(* CODESYS project METIS_CRYO.library
   Version: 0.1.1
   Title: METIS Cryo PLC
   Author: Muhammad Salman
   Placeholder: METIS Cryo PLC
   Company: KU Leuven

Project tree, tasks and I/O mapping:
  libraries: CmpBitmapPool, * (System); ESO Cryo HMI Library, * (ESO); ESO LDC Comm Common Library, * (ESO); ESO LDC Comm Tcp Library, * (ESO); ESO LDC Control Library, * (ESO); ESO LDC Cryo Library, * (ESO); ESO LDC Timer Library, * (ESO); FloatingPointUtils, * (System); METIS CCU, * (KU Leuven); METIS Fuse Library, * (KU Leuven); Recipe Management, * (System); Tc2_ControllerToolbox, * (Beckhoff Automation GmbH); Tc2_Standard, * (Beckhoff Automation GmbH); Tc2_System, * (Beckhoff Automation GmbH); Tc2_Utilities, * (Beckhoff Automation GmbH); Tc2_XmlDataSrv, * (Beckhoff Automation GmbH); Tc3_Module, * (Beckhoff Automation GmbH); VisuDialogs, * (System); VisuSymbols, * (System)
  DUTs/
    Enumerators/
      Actuators/
      Ctrl_Valves/
        data type E_METIS_CRYO_CTRL_VALVE_STATE
        data type E_METIS_CRYO_CTRL_VALVE_TYPE
      Heaters/
        data type E_METIS_CRYO_HEATER_STATE
        data type E_METIS_CRYO_HEATER_TYPE
        data type E_METIS_PWM_HEATER_CTRL
      LN2_Level/
        data type E_LN2_LEVEL_CTRL_STATE
      Routines/
        Anti_Fogging/
          data type E_ANTI_FOGGING_MODE
          data type E_MET_CRYO_ANTI_FOGGING_STATE
        Cool_Down/
          data type E_MET_CRYO_COOLDOWN_PRESSURES
          data type E_MET_CRYO_COOLDOWN_STATE
          data type E_MET_CRYO_COOLDOWN_SYS_STATE
          data type E_MET_CRYO_COOLDOWN_VALVES
          data type E_MET_CRYO_LN2_FILLING_STATE
        Re_Generation/
          data type E_MET_CRYO_RE_GENERATION_STATE
        Venting/
          data type E_MET_CRYO_VENTING_PRESSURES
          data type E_MET_CRYO_VENTING_STATE
          data type E_MET_CRYO_VENTING_SYS_STATE
          data type E_MET_CRYO_VENTING_VALVES
        WarmUp/
          data type E_MET_CRYO_WARMUP_STATE
      Sensors/
        Base_Sensor/
          data type E_METIS_SENSOR_SOURCE
          data type E_METIS_SENSOR_TYPE
        LN2_Level_Sensor/
          data type E_METIS_CRYO_LN2_SENSOR_LEVELS
        Temperature Sensor/
          data type E_METIS_LAKE_SHORE_TYPE
          data type E_METIS_TEMP_VOTE_METHOD
      System/
        data type E_METIS_CRYO_CTRL_CMD
        data type E_METIS_CRYO_CTRL_STATE
    Structures/
      Actuators/
      Base_Sensor/
        data type T_METIS_SENSOR_BASE_STATUS
      Ctrl_Valves/
        data type T_METIS_CTRL_VALVE_CFG
        data type T_METIS_CTRL_VALVE_CTRL
        data type T_METIS_CTRL_VALVE_IO_ANTI_FOG_BLOWER
        data type T_METIS_CTRL_VALVE_IO_IMG_CFO_PRECOOLING
        data type T_METIS_CTRL_VALVE_STAT
      Error_Handeling/
        data type T_METIS_CRYO_ERROR_STATUS
      Heaters/
        METIS_HEATER/
          data type T_METIS_HEATER_CFG
          data type T_METIS_HEATER_CTRL
          data type T_METIS_HEATER_IO_CPAU60
          data type T_METIS_HEATER_IO_CXWUI60
          data type T_METIS_HEATER_IO_EL95X1
          data type T_METIS_HEATER_IO_PWM
          data type T_METIS_HEATER_STAT
        data type T_METIS_CRYO_HEATER_CTRL
        data type T_METIS_CRYO_HEATER_STATUS
      LN2_Level_Ctrl/
        data type T_LN2_LEVEL_CTRL_CFG
        data type T_LN2_LEVEL_CTRL_CTRL
      PID_Control/
        Generic/
          data type E_METIS_CTRL_MODE
          data type E_METIS_CTRL_SETPOINT_SWITCH
          data type T_METIS_CTRL_LOOP_CFG
          data type T_METIS_CTRL_LOOP_CTRL
          data type T_METIS_CTRL_LOOP_STAT
          text list TEXTLIST_METIS_CTRL_MODE
        data type T_METIS_CTRL_BASE_CFG
        data type T_METIS_CTRL_BASE_CTRL
        data type T_METIS_CTRL_BASE_STAT
      RAMP/
        data type T_METIS_CTRL_RAMP_CTRL
        data type T_METIS_CTRL_RAMP_STAT
      Routines/
        Anti_Fogging/
          data type T_MET_CRYO_ANTI_FOGGING_CTRL
          data type T_MET_CRYO_ANTI_FOGGING_STAT
        Cool_Down/
          data type T_MET_CRYO_COOLDOWN_CFG
          data type T_MET_CRYO_COOLDOWN_CTRL
          data type T_MET_CRYO_COOLDOWN_STAT
          data type T_MET_CRYO_COOLDOWN_SYS_INPUT
          data type T_MET_CRYO_COOLDOWN_SYSTEM_STATUS
        Evacuation/
          data type T_MET_CRYO_EVACUATION_CTRL
          data type T_MET_CRYO_EVACUATION_STAT
        Re_Generation/
          data type T_MET_CRYO_RE_GENERATION_CTRL
          data type T_MET_CRYO_RE_GENERATION_STAT
        Venting/
          data type T_MET_CRYO_VENTING_CFG
          data type T_MET_CRYO_VENTING_CTRL
          data type T_MET_CRYO_VENTING_STAT
          data type T_MET_CRYO_VENTING_SYS_INPUT
          data type T_MET_CRYO_VENTING_SYSTEM_STATUS
        WarmUp/
          data type T_MET_CRYO_WARMUP_CTRL
          data type T_MET_CRYO_WARMUP_STAT
      Sensors/
        LN2_Level_Sensor/
          data type T_METIS_CRYO_LN2_LEVEL_CFG
          data type T_METIS_CRYO_LN2_LEVEL_STATUS
      System/
        data type T_METIS_CRYO_CFG
        data type T_METIS_CRYO_CTRL
        data type T_METIS_CRYO_DEBUG
        data type T_METIS_CRYO_EVENTS
        data type T_METIS_CRYO_INTERLOCKS
        data type T_METIS_CRYO_STAT
        data type T_METIS_CRYO_TRIGGERS
      Temp_Sensor/
        data type T_METIS_DT670_TEMP_SENSOR_STATUS
      Temp_Voter/
        data type T_HMI_METIS_TEMP_VOTER_CTRL
        data type T_HMI_METIS_TEMP_VOTER_STAT
        data type T_METIS_CRYO_TEMP_VOTE_STATUS
        data type T_METIS_TEMP_VOTE_CFG
        data type T_METIS_TEMP_VOTERS_CTRL
      Temperature/
        data type E_ALL_METIS_TEMPERATURES
        data type T_METIS_TEMPERATURE_STATUS
  GVLs/
  HMI/
    DUTs/
      Cryo_Devices/
        Temperatures/
          data type E_HMI_TEMP_TABS
        data type E_HMI_PUMPS_TABS
      Subsystems/
        CFO/
          data type E_HMI_CFO_TABS
        CRY/
          Components/
            data type E_HMI_CRY_HEATER_TABS
            data type E_HMI_CRY_TC_TABS
          data type E_HMI_CRY_TABS
        ICS/
          data type E_HMI_ICS_TABS
        IMG/
          Components/
            data type E_HMI_IMG_HEATER_TABS
            data type E_HMI_IMG_TC_TABS
          data type E_HMI_IMG_TABS
        LMS/
          data type E_HMI_LMS_TABS
        SCA/
          Components/
            data type E_HMI_SCA_HEATER_TABS
            data type E_HMI_SCA_TC_TABS
          data type E_HMI_SCA_TABS
      System/
        data type E_HMI_TABS
      Util/
        data type E_HMI_COLORS
        data type E_HMI_VOTER_TABS
        data type T_ECAT_MODULE
        data type T_HMI_COLORS
    POUs/
      Cryo-Routines/
        Anti-Fogging/
          function block FB_HMI_ANTI_FOGGING [ST]
        Cool-Down/
          function block FB_HMI_COOL_DOWN [ST]
        Evacuation/
          function block FB_HMI_EVACUATION [ST]
        Power-Outage/
          function block FB_HMI_POWER_OUTAGE [ST]
        Regeneration/
          function block FB_HMI_REGENERATION [ST]
        Venting/
          function block FB_HMI_VENTING [ST]
        Warm-Up/
          function block FB_HMI_WARM_UP [ST]
      Devices/
        Cabinets/
          function block FB_HMI_CABINETS [ST]
          function block FB_HMI_CCU [ST]
        Control_Loops/
          function block FB_HMI_CONTROL_LOOPS [ST]
          function block FB_HMI_METIS_CTRL_TEMPERATURE [ST]
        Control_Units/
          function block FB_HMI_CONTROL_UNITS [ST]
        Coolers/
          function block FB_HMI_COOLERS [ST]
        Detectors/
          function block FB_HMI_DETECTORS [ST]
        Heaters/
          function block FB_HMI_HEATERS [ST]
          function block FB_HMI_METIS_HEATER [ST]
        Lakeshores/
          function block FB_HMI_LAKESHORE [ST]
        Pressures/
          function block FB_HMI_PRESSURES [ST]
        Pumps/
          function block FB_HMI_PUMPS [ST]
          function block FB_HMI_RP_BRANCH_A [ST]
          function block FB_HMI_RP_BRANCH_B [ST]
          function block FB_HMI_TP_BRANCH_A [ST]
          function block FB_HMI_TP_BRANCH_B [ST]
        RH/
          function block FB_HMI_METIS_RH_SENSOR [ST]
        Temperatures/
          Components/
            function block FB_HMI_TEMP_VOTERS [ST]
          function block FB_HMI_TEMPERATURES [ST]
        Valves/
          function block FB_HMI_VALVES [ST]
        Voters/
          function block FB_HMI_VOTER [ST]
        function block FB_HMI_DEVICES [ST]
      Events/
        function block FB_HMI_EVENTS [ST]
      ICS_Interlocks/
        function block FB_HMI_ICS_INTERLOCKS [ST]
      Services/
        Status/
          function F_HMI_BUSY_TO_COLOR [ST]
          function F_HMI_HEALTH_BUSY_TO_COLOR [ST]
          function F_HMI_HEALTH_TO_COLOR [ST]
          function block FB_HMI_BUSY_STATUS [ST]
          function block FB_HMI_HEALTH_STATUS [ST]
          function block FB_HMI_STATUS [ST]
        function block FB_HMI_SERVICES [ST]
        function block FB_HMI_SERVICES_TIME [ST]
      Subsystems/
        CFO/
          Components/
            function block FB_HMI_CFO_HEATERS [ST]
            function block FB_HMI_CFO_TCTRL [ST]
            function block FB_HMI_CFO_TEMPERATURES [ST]
            function block FB_HMI_CFO_VOTERS [ST]
          function block FB_HMI_CFO [ST]
        CRY/
          Components/
            function block FB_HMI_CRY_HEATERS [ST]
            function block FB_HMI_CRY_LN2CTRL [ST]
            function block FB_HMI_CRY_RH [ST]
            function block FB_HMI_CRY_TCTRL [ST]
            function block FB_HMI_CRY_TEMPERATURES [ST]
            function block FB_HMI_CRY_VOTERS [ST]
          function block FB_HMI_CRY [ST]
        ICS/
          function block FB_HMI_ICS [ST]: M_UpdateConfigsColor
        IMG/
          Components/
            function block FB_HMI_IMG_HEATERS [ST]
            function block FB_HMI_IMG_TCTRL [ST]
            function block FB_HMI_IMG_TEMPERATURES [ST]
            function block FB_HMI_IMG_VOTERS [ST]
          function block FB_HMI_IMG [ST]
        LMS/
          Components/
            function block FB_HMI_LMS_HEATERS [ST]
            function block FB_HMI_LMS_TCTRL [ST]
            function block FB_HMI_LMS_TEMPERATURES [ST]
            function block FB_HMI_LMS_VOTERS [ST]
          function block FB_HMI_LMS [ST]
        SCA/
          Components/
            function block FB_HMI_SCA_HEATERS [ST]
            function block FB_HMI_SCA_TCTRL [ST]
            function block FB_HMI_SCA_TEMPERATURES [ST]
            function block FB_HMI_SCA_VOTERS [ST]
          function block FB_HMI_SCA [ST]
      Util/
        Button/
          function block FB_HMI_BUTTON [ST]: FB_init, M_SetIconName
        Component/
          function block FB_HMI_COMPONENT [ST]: M_UpdateStatusColor
        Functions/
          function F_GetConnectionColor [ST]
          function F_GetConnectionString [ST]
        function block FB_HMI_BACK [ST]
        function block FB_HMI_CRYO_SIM [ST]
    VISUs/
      Cryo_Devices/
        Cabinets/
          visualisation VISU_HMI_CABINETS
        Control_Loops/
          visualisation VISU_HMI_CONTROL_LOOPS
        Control_Units/
          visualisation VISU_HMI_CONTROL_UNITS
        Coolers/
          visualisation VISU_HMI_COOLERS
        Detectors/
          visualisation VISU_HMI_DETECTORS
        Heaters/
          visualisation VISU_HMI_HEATERS
        Pressures/
          visualisation VISU_HMI_PRESSURES
        Pumps/
          visualisation VISU_HMI_PUMPS
          visualisation VISU_HMI_RP_BRANCH_A
          visualisation VISU_HMI_RP_BRANCH_B
          visualisation VISU_HMI_TP_BRANCH_A
          visualisation VISU_HMI_TP_BRANCH_B
        Temperatures/
          Components/
            visualisation VISU_HMI_SYSTEM_VOTERS
          visualisation VISU_HMI_TEMPERATURES
        Valves/
          visualisation VISU_HMI_VALVES
        visualisation VISU_HMI_DEVICES_DIALOG
      Cryo-Routines/
        Anti-Fogging/
          visualisation VISU_HMI_ANTI_FOGGING
        Cool-Down/
          visualisation VISU_HMI_COOL_DOWN
        Evacuation/
          visualisation VISU_HMI_EVACUATION
        Power-Outage/
          visualisation VISU_HMI_POWER_OUTAGE
        Regeneration/
          visualisation VISU_HMI_REGENERATION
          visualisation VISU_REGENERATION_CTRL
          visualisation VISU_SORPTION_HEATER
          visualisation VISU_SORPTION_TEMP_VOTE
        Venting/
          visualisation VISU_HMI_VENTING
        Warm-Up/
          visualisation VISU_HMI_WARM_UP
      Events/
        visualisation VISU_HMI_EVENTS
      GUIs/
        visualisation GUI_LN2_LEVEL_CTRL
        visualisation GUI_MANUAL_CONTROL
        visualisation GUI_METIS_EVACUATION
        visualisation VISU_HMI_FUSE_HMI
      Home/
        visualisation VISU_HMI_HOME
      ICS_Interlocks/
        visualisation VISU_HMI_ICS_INTERLOCKS
      Services/
        visualisation VISU_HMI_SERVICES
      SIM_GUIs/
        visualisation GUI_Pressures_1
        visualisation GUI_SIM_PRESSURES
        visualisation GUI_SIM_SYSTEM_STATE
        visualisation GUI_SIM_TEMPERATURES
        visualisation VISU_SIM_PRESS_AND_TEMPS
      Subsystems/
        CFO/
          Components/
          visualisation VISU_HMI_CFO
        CRY/
          Components/
            visualisation VISU_HMI_CRY_HEATERS
            visualisation VISU_HMI_CRY_LN2_LEVEL_CONTROL
            visualisation VISU_HMI_CRY_RH
            visualisation VISU_HMI_CRY_TCTRL
            visualisation VISU_HMI_CRY_TEMPERATURES
            visualisation VISU_HMI_CRY_VOTERS
          visualisation VISU_HMI_CRY
        ICS/
          Components/
            visualisation VISU_HMI_ICS_CCU_CONFIGS
            visualisation VISU_HMI_ICS_CCUS_CONFIGS
          visualisation VISU_HMI_ICS
        IMG/
          Components/
            visualisation VISU_HMI_IMG_HEATERS
            visualisation VISU_HMI_IMG_TC
            visualisation VISU_HMI_IMG_TEMPERATURES
            visualisation VISU_HMI_IMG_VOTERS
          visualisation VISU_HMI_IMG
        LMS/
          visualisation VISU_HMI_LMS
        SCA/
          Components/
            visualisation VISU_HMI_SCA_HEATERS
            visualisation VISU_HMI_SCA_TC
            visualisation VISU_HMI_SCA_TEMPERATURES
            visualisation VISU_HMI_SCA_VOTERS
          visualisation VISU_HMI_SCA
      Templates/
        visualisation ARCHIVED_TEMPLATE_MAIN_FSM_1
        visualisation GUI_EVAC_BRANCH_A_1
        visualisation GUI_Events
        visualisation GUI_RP_PUMPS
        visualisation GUI_TEMPLATE_LAKESHORE_336_TCP
        visualisation GUI_TP_PUMPS
        image pool ImagePool_1
        visualisation Sim_LN2_Ctrl_inputs
        visualisation TEMPLATE_AMBIENT_PRESSURE_READING
        visualisation TEMPLATE_BACKGROUND_LEVEL_2
        visualisation TEMPLATE_BACKGROUND_LEVEL_3
        visualisation TEMPLATE_BINARY_VALVES
        visualisation TEMPLATE_CRYO_SENSOR_TEMPERATURE
        visualisation TEMPLATE_EVACUATION
        visualisation TEMPLATE_HEATER_CPAU60
        visualisation TEMPLATE_HEATER_CXWUI60
        visualisation TEMPLATE_HEATER_PWM_CTRL
        visualisation TEMPLATE_LN2_LEVEL_SENSOR_AND_CTRL
        visualisation TEMPLATE_MAIN_FSM
        visualisation TEMPLATE_METIS_CMD_OVERRIDE
        visualisation TEMPLATE_METIS_CONTROL_VALVE
        visualisation TEMPLATE_METIS_CRYO_CPA
        visualisation TEMPLATE_METIS_CRYO_CPAU60_PID_CTRL
        visualisation TEMPLATE_METIS_CRYO_PWM_PID_CTRL
        visualisation TEMPLATE_METIS_CTRL_TEMPERATURE
        visualisation TEMPLATE_METIS_CTRL_TEMPERATURE_MPIA
        visualisation TEMPLATE_METIS_CTRL_TEMPERATURE_SIMPLIFIED
        visualisation TEMPLATE_METIS_HEATER
        visualisation TEMPLATE_METIS_HEATER_SIMPLIFIED
        visualisation TEMPLATE_PRESSURE_READING
        visualisation TEMPLATE_RESET_VALVES
        visualisation TEMPLATE_TEMP_SENSOR_VALUE_ONLY
        visualisation TEMPLATE_TEMPERATURE_VOTE
      Util/
        Button/
          image pool VISU_HMI_BUTTON_IMAGES
          visualisation VISU_HMI_ROUTINES_BUTTON
          visualisation VISU_HMI_SUBSUBSYSTEM_BUTTON
          visualisation VISU_HMI_SUBSYSTEM_BUTTON
          visualisation VISU_HMI_SYSTEM_BUTTON
        image pool ICONS_IMAGE_POOL
    program PRG_HMI [ST]: M_TrackPreviousTab, M_UpdateStatus
    visualisation VISU_HMI
  00000000-0000-0000-0000-000000000000|IMAGES\Evacuation_schematics.png
  00000000-0000-0000-0000-000000000000|IMAGES\METIS_Cryo_FSM.png
  00000000-0000-0000-0000-000000000000|HMI\Images\Button\home.png
  00000000-0000-0000-0000-000000000000|HMI\Images\Button\cover.png
  00000000-0000-0000-0000-000000000000|HMI\Images\Button\m1.png
  00000000-0000-0000-0000-000000000000|HMI\Images\Button\m3.png
  00000000-0000-0000-0000-000000000000|HMI\Images\Button\services.png
  00000000-0000-0000-0000-000000000000|HMI\Images\Button\telemetry.png
  00000000-0000-0000-0000-000000000000|HMI\Images\Button\m2.png
  00000000-0000-0000-0000-000000000000|HMI\Images\Button\hydraulics.png
  00000000-0000-0000-0000-000000000000|HMI\Images\Button\safety.png
  00000000-0000-0000-0000-000000000000|HMI\Images\Button\axes.png
  00000000-0000-0000-0000-000000000000|HMI\Images\Button\dome.png
  00000000-0000-0000-0000-000000000000|HMI\Images\Button\Events.png
  00000000-0000-0000-0000-000000000000|HMI\Images\Button\subsystems.png
  00000000-0000-0000-0000-000000000000|HMI\Images\Button\interlock.png
  00000000-0000-0000-0000-000000000000|Images\metis_logo_white.png
  00000000-0000-0000-0000-000000000000|Images\metis_logo_color.png
  HMIWrapperFBs/
    function block FB_METIS_HMI_CRYO_TEMPERATURE_VOTE [ST]: M_ProcessInput, M_UpdateStatus
  IMAGES/
    Evacuation_schematics.png
  POUs/
    Control/
      Control/
        function block FB_METIS_CTRL_BASE [ST]: M_CheckErrors, M_Configure, M_ExecuteController, M_Read_Write_Config, M_Set_PID_Parameters, M_SetAutoMode, M_SetEngMode, M_SetManualMode, M_SetPermissionMode, M_SetRamp
        function block FB_METIS_CTRL_RAMP_GENERATOR [ST]: M_Configure, M_ExecuteController
        function block FB_METIS_CTRL_TEMPERATURE [ST]: M_ConfigReadingFinished, M_Configure, M_ExecuteController, M_ExecuteModes, M_Read_Write_Config, M_Set_SetPoint, M_SetDisable, M_SetEnable, M_Startup, M_UpdateAlarms, M_UpdateStatus, M_UpdateTempPointers
        function block FB_PWM_PID_CTRL [ST]
      Process/
        function block FB_FT1_SIM_PROCESS [ST]
      TCtrl/
        function block FB_METIS_TCTRL [ST]
    Devices/
      AmbientPressure/
        function block FB_METIS_AMBIENT_PRESSURE_SENSOR [ST]: M_SetStatus, M_SetStatus_CMR_361, M_SetStatus_MIPA_015A, M_SetStatus_PKR_250, M_SetStatus_PKR_360, M_SetStatus_WRG_D_NW25
      Base_Sensor/
        function block FB_METIS_SENSOR_BASE [ST]: M_GetRamp, M_ReadSensor, M_SetStatus, M_SetStatus_LS240
      CCU/
        function block FB_METIS_CCUS [ST]: M_Configure
      Control_Valves_Ctrl/
        function block FB_METIS_CONTROL_VALVE [ST]: M_Activity_Valve_Alarm, M_Activity_Valve_None, M_Activity_Valve_Normal, M_Configure, M_GetError, M_IsValveInError, M_Read_Write_Config, M_ReadInputs, M_ScaleInput, M_ScaleOutput, M_SetCtrlOutput, M_SetDisable, M_SetEnable, M_SetManualDisable, M_SetManualEnable, M_SetMode, M_SetStatus, M_UpdateActive, M_UpdateAlarms
      DigitalOutput/
        function block FB_METIS_DO [ST]: M_Configure, M_UpdateStatus
        data type T_METIS_DO_CTRL
        data type T_METIS_DO_STAT
      Heaters/
        Heater_Ctrl/
          function block FB_HEATER_CPAU60 [ST]: bIsActive, bIsInError, bIsNotActive, lrHeaterPower, M_Activate, M_Configure, M_DeActivate, M_GetHeaterPower, M_ReadInputs, M_ScaleInput, M_ScaleOutput, M_SetCtrlOutput, M_SetHeaterPower, M_SetManualInputFlag, M_SetStatus
          function block FB_HEATER_CXWUI60 [ST]: bIsActive, bIsInError, bIsNotActive, lrHeaterPower, M_Activate, M_Configure, M_DeActivate, M_GetHeaterPower, M_ReadInputs, M_ScaleInput, M_ScaleOutput, M_SetCtrlOutput, M_SetHeaterPower, M_SetManualInputFlag, M_SetStatus
          function block FB_HEATER_PWM [ST]: bIsActive, bIsInError, bIsNotActive, lrHeaterPower, M_Activate, M_DeActivate, M_GetHeaterPower, M_ReadInputs, M_ScaleInput, M_ScaleOutput, M_SetCtrlOutput, M_SetHeaterPower, M_SetManualInputFlag, M_SetStatus
          function block FB_METIS_HEATER [ST]: M_Configure, M_isHeaterInError, M_Read_Write_Config, M_ReadInputs, M_ScaleInput, M_ScaleOutput, M_SetCtrlOutput, M_SetDisable, M_SetEnable, M_SetMode, M_SetStatus, M_UpdateAlarms
          interface I_Heater: bIsActive, bIsInError, bIsNotActive, lrHeaterPower, M_Activate, M_DeActivate
        function block FB_METIS_HEATERS [ST]: M_ExecuteControllers
      LakeShore_336/
        function block FB_METIS_LAKESHORE_336_TCP [ST]: M_Configure, M_GetCommInitialised, M_GetCommStatus, M_SetTemperatureOutputs, M_UpdateStatus
        function block FB_METIS_LAKESHORES [ST]
      LN2_Level_Ctrl/
        function block FB_METIS_CRYO_LN2_LEVEL_CTRL [ST]: M_Activity_CheckPreConditions, M_Activity_EarlyRefilling, M_Activity_ErrorHandeling, M_Activity_Level_Monitoring, M_Check_LN2_Level, M_Configure, M_ExecuteControllers, M_FillingControl, M_HandleEvents, M_Read_Write_Config, M_ReadSensors, M_Reset, M_ResetValve, M_Set_LN2FillingFlag, M_StateMachine, M_UpdateAlarms, M_UpdateStatus
      LN2_Level_Sensor/
        function block FB_LN2_LEVEL_PT100_SENSOR [ST]
        function block FB_METIS_CRYO_LN2_SENSOR [ST]: M_ReadSensors, M_SetHeatersOutput, M_SetOutput, M_SetStatus
      PTC Cooler/
        function block FB_METIS_CRYO_CPA [ST]: M_CompressorRunning, M_HighPressureFlag, M_HighTemperatureFlag
      RH_Sensor/
        function block FB_METIS_RH [ST]
        function block FB_METIS_RH_DEWPOINT_CALC [ST]
        function block FB_METIS_RH_SENSOR [ST]: M_ReadSensor, M_SetStatus
        data type T_METIS_RH_SENSOR_STAT
      Temp_Sensor/
        function block FB_METIS_TEMP_SENSOR_DT670 [ST]: M_GetRamp, M_ReadSensor, M_SetSensorStatus_DT670_LS240, M_SetSensorStatus_DT670_LS336, M_SetSensorStatus_DT670_Ramp, M_SetSensorStatus_DT670_Voter, M_SetStatus, M_SetTemperature
        function block FB_SIM_TEMP_SENSOR_DT670 [ST]: M_Configure, M_ExecuteController
      Temp_Voter/
        function block FB_METIS_VOTER [ST]: bTempNotValid, bTempValid, lrRamp, lrTempK, M_ConfigReadingFinished, M_Configure, M_GetRamp, M_Read_Write_Config, M_SetPermissionMode, M_SetStatus, M_SetStatus_Average, M_SetStatus_FirstValid, M_SetStatus_Highest_Temperature, M_SetStatus_Lowest_Temperature, M_SetStatus_Median, M_SetStatus_XooY, M_UpdateAlarms, M_UpdateTempPointers
        function block FB_METIS_VOTER_COPY_for_new_HMI [ST]: bTempNotValid, bTempValid, lrRamp, lrTempK, M_ConfigReadingFinished, M_Configure, M_GetRamp, M_Read_Write_Config, M_SetPermissionMode, M_SetStatus, M_SetStatus_Average, M_SetStatus_FirstValid, M_SetStatus_Highest_Temperature, M_SetStatus_Lowest_Temperature, M_SetStatus_Median, M_SetStatus_XooY, M_UpdateTempPointers
        function block FB_METIS_VOTERS [ST]: M_ProcessHmi, M_ReadSensors
      Temperature/
        function block FB_METIS_TEMPERATURE [ST]
        function block FB_METIS_TEMPERATURES [ST]: M_ConfigSimTemperatures, M_Configure, M_GetTempSensorIndex, M_IsIgnoredTemperature, M_MaxMinAvrgTemperatures, M_ReadSensors, M_SetTemperatureSensor, M_UpdatePointer, M_UpdatePointers
    Functions/
      function F_TIME_HHMMSS [ST]
      function F_TON_TO_TIME_STRING [ST]
    Routines/
      AntiFogging/
        function block FB_METIS_CRYO_ANTI_FOGGING [ST]: M_Activity_AirBlowing, M_Activity_Alarm_Condition, M_Activity_Check_Preconditions, M_Activity_Error_Handling, M_Activity_Finished, M_Activity_Heating, M_Activity_None, M_Activity_Standard_Operation, M_Activity_Start_Anti_Fogging, M_Configure, M_Evaluate_DewPoint_State, M_ExecuteControllers, M_HandleEvents, M_SetError, M_Start_AntiFogging, M_StateMachine, M_Stop_AntiFogging, M_UpdateStatus
      CabinetControl/
        function block FB_METIS_CABINET_CTRL [ST]
      CoolDown/
        function block FB_METIS_CRYO_COOL_DOWN [ST]: M_Activity_Check_Preconditions, M_Activity_Cold_State, M_Activity_Cool_Down_Finished, M_Activity_Error_Handling, M_Activity_Finished, M_Activity_Keep_Cooling, M_Activity_None, M_Activity_Start_Cool_Down, M_Activity_Start_LN2_Filling, M_Activity_Start_PTCs, M_Activity_Start_Temp_Ctrl_PTC, M_Activity_Stop_LN2_Filling, M_Activity_Stop_PTCs, M_Activity_Stopping_Cool_Down, M_Check_Is_ReadyForOperation, M_Check_LN2_Filling_Status, M_Check_PTCs_Heater_Ctrl_Status, M_Check_PTCs_Status, M_Configure, M_ExecuteControllers, M_Get_ReadyForOperations, M_HandleEvents, M_HandleInterlocks, M_Manage_Early_Refilling, M_PermitEvacuationStop, M_ReadSensors, M_ResetValves, M_SetError, M_Simulated_Sens_Acts, M_Standalone_LN2_Filling, M_StateMachine, M_Stop_PTCs_During_WarmUP, M_UpdateStatus
      Evacuation/
        function block FB_CRYO_EVAC_BRANCH_A [ST]: M_Configure, M_ExecuteControllers, M_HandleInterlocks, M_ResetValves
        function block FB_CRYO_EVAC_BRANCH_B [ST]: M_Configure, M_ExecuteControllers, M_HandleInterlocks, M_ResetValves
        function block FB_METIS_CRYO_EVAC [ST]: M_AreAnyPumpsRunning, M_AreRoughingPumpRunning, M_AreTurboPumpsRunning, M_CheckBranchError, M_Configure, M_ExecuteControllers, M_HandleEvents, M_HandleInterlocks, M_ResetValves, M_SetAuto, M_SetError, M_Start_Evacuation, M_Stop_Evacuation, M_UpdateStatus
      PowerOutage/
        function block FB_METIS_CRYO_POWER_OUTAGE [ST]
      Regeneration/
        function block FB_METIS_CRYO_REGENERATION [ST]: M_Activity_Check_Preconditions, M_Activity_CoolDownSP, M_Activity_ErrorHandeling, M_Activity_Finished, M_Activity_KeepHeating, M_Activity_None, M_Activity_StartHeating, M_Configure, M_ExecuteControllers, M_HandleEvents, M_PermitEvacuationStop, M_SetError, M_StateMachine, M_UpdateStatus
      StopPowerOutage/
        function block FB_METIS_CRYO_STOP_POWER_OUTAGE [ST]
      Venting/
        function block FB_METIS_CRYO_VENTING [ST]: M_Activity_Check_Preconditions, M_Activity_ClosingValve, M_Activity_Error_Handling, M_Activity_None, M_Activity_OpeningValve, M_Activity_Prepare_For_Venting, M_Activity_Start_Venting, M_Activity_Stop_Venting, M_Activity_Venting_InProgress, M_AreVentingValvesClosed, M_Close_Venting_Valves, M_Configure, M_ExecuteControllers, M_HandleEvents, M_HandleInterlocks, M_IsVentingFinishedSuccessfully, M_Open_Venting_Valves, M_ReadSensors, M_ResetValves, M_SetError, M_StateMachine, M_UpdateStatus
      WarmUP/
        function block FB_METIS_CRYO_WARM_UP [ST]: M_Activity_Check_Preconditions, M_Activity_Error_Handling, M_Activity_Finished, M_Activity_Keep_Ramping_Up_Detectors, M_Activity_Keep_Warming_Up, M_Activity_None, M_Activity_Ramp_Up_Detectors_2, M_Activity_Start_Ramp_Up_CFO, M_Activity_Start_Ramp_Up_Detectors_1k, M_Activity_Start_Ramp_Up_IMG, M_Activity_Start_Ramp_Up_LMS, M_Activity_Start_Ramp_Up_Radiation_Shields, M_Activity_Start_Ramp_Up_SCAO, M_Activity_Start_Warm_Up, M_Activity_Stop_PTCs, M_Activity_Stopping_Warm_Up, M_AreWarmUpHeaterActive, M_CheckTCErrors, M_Configure, M_HandleEvents, M_HandleInterlocks, M_PermitEvacuationStop, M_PermitVenting, M_SetError, M_StateMachine, M_UpdateStatus
    Services/
      function block FB_SERVICES [ST]
    Simulation/
      function block FB_SIM_LN2_LEVEL_VALVES [ST]
      function block FB_SIM_LN2_SENSOR [ST]
      function block FB_SIM_PRE_COOLING_VALVES [ST]
      function block FB_SIM_REGENERATION [ST]
      function block FB_SIM_VENTING_VALVES [ST]
    System/
      function block FB_METIS_CRYO_CTRL [ST]: M_Activity_Cold_State, M_Activity_Cooling_Down_State, M_Activity_Error_State, M_Activity_None, M_Activity_Partial_Vacuum_State, M_Activity_Partially_Cold_State, M_Activity_Stabilize_Cryostat_Conditions, M_Activity_Venting, M_Activity_Warm_Press_State, M_Activity_Warm_Up_State, M_Activity_Warm_Vacuum_State, M_CheckDetectorsSafety, M_CheckDetectorTempStability, M_CheckForCommands, M_CheckForSensorErrors, M_CheckLakeshoreCommand, M_CheckVacuum, M_Configure, M_ExecuteControllers, M_GetHighestTemperature, M_GetLowestTemperature, M_GetState, M_HMI_Screen_Control, M_ProcessHmi, M_ReadSensors, M_SafetyCheck, M_SetError, M_SetStatus, M_StateMachine, M_SysLog, M_UpdatePressureStates, M_UpdateStatus
    XML_Cfg_Read_Write/
      function block FB_READ_WRITE_CAB_COOLING_CONFIG [ST]
      function block FB_READ_WRITE_CAB_POWER_CONFIG [ST]
      function block FB_READ_WRITE_CONFIG_BASE [ST]: bIsReading, bIsWriting, M_ClearReadingDoneFlag, M_ClearWritingDoneFlag, M_Configure, M_GetErrorString, M_ReadConfiguration, M_WriteConfiguration
      function block FB_READ_WRITE_CONTROL_VALVE_CONFIG [ST]
      function block FB_READ_WRITE_HEATER_CONFIG [ST]
      function block FB_READ_WRITE_LN2_LEVEL_CONTROL_CONFIG [ST]
      function block FB_READ_WRITE_METIS_CTRL_DT670_CFG [ST]
      function block FB_READ_WRITE_TEMP_CONTROL_CONFIG [ST]
      function block FB_READ_WRITE_TEMP_VOTE_CONFIG [ST]
    program MAIN [ST]
  text list GlobalTextList
*)

// DUTs/Enumerators/Ctrl_Valves/E_METIS_CRYO_CTRL_VALVE_STATE
{attribute 'qualified_only'}
{attribute 'strict'}
TYPE E_METIS_CRYO_CTRL_VALVE_STATE :
(
	OFF := 0,
	STARTING,
	ON,
	STOPPING,
	ERROR
);
END_TYPE

// DUTs/Enumerators/Ctrl_Valves/E_METIS_CRYO_CTRL_VALVE_TYPE
{attribute 'qualified_only'}
{attribute 'strict'}
TYPE E_METIS_CRYO_CTRL_VALVE_TYPE :
(	 NONE := 0,
	 ANTI_FOG_BLOWER,
	 PRE_COOLING_IMG_CFO
);
END_TYPE

// DUTs/Enumerators/Heaters/E_METIS_CRYO_HEATER_STATE
{attribute 'qualified_only'}
{attribute 'strict'}
TYPE E_METIS_CRYO_HEATER_STATE :
(
	OFF := 0,
	STARTING,
	ON,
	STOPPING,
	ERROR
);
END_TYPE

// DUTs/Enumerators/Heaters/E_METIS_CRYO_HEATER_TYPE
{attribute 'qualified_only'}
{attribute 'strict'}
TYPE E_METIS_CRYO_HEATER_TYPE :
(	 NONE := 0,
	 CPAU60 ,
	 CXWUI60,
	 PWM_DETECTOR,
	 PWM_SORPTION,
	 PWM_WINDOW,
     EL95X1
);
END_TYPE

// DUTs/Enumerators/Heaters/E_METIS_PWM_HEATER_CTRL
{attribute 'qualified_only'}
{attribute 'strict'}
TYPE E_METIS_PWM_HEATER_CTRL :
(
	SorptionPump_Heater_Ctrl := 0,
	Detector_Heater_Ctrl
);
END_TYPE

// DUTs/Enumerators/LN2_Level/E_LN2_LEVEL_CTRL_STATE
{attribute 'qualified_only'}
{attribute 'strict'}
TYPE E_LN2_LEVEL_CTRL_STATE :
(
	OFF := 0,
	CHECK_PRECONDITIONS,
	EARLY_REFILLING,
	LEVEL_MONITORING,
	ERROR
);
END_TYPE

// DUTs/Enumerators/Routines/Anti_Fogging/E_ANTI_FOGGING_MODE
{attribute 'qualified_only'}
{attribute 'strict'}
TYPE E_ANTI_FOGGING_MODE :
(
	PURGING := 0,
	HEATING,
	PURGING_AND_HEATING
);
END_TYPE

// DUTs/Enumerators/Routines/Anti_Fogging/E_MET_CRYO_ANTI_FOGGING_STATE
{attribute 'qualified_only'}
{attribute 'strict'}
TYPE E_MET_CRYO_ANTI_FOGGING_STATE :
(
	NONE := 0, 
	CHECK_PRECONDITIONS := 1, 
	START_ANTI_FOGGING,
	STANDARD_OPERATION, 
	AIR_BLOWING, 
	HEATING,
	ALARM_CONDITION, 
	FINISHED, 
	ERROR
);
END_TYPE

// DUTs/Enumerators/Routines/Cool_Down/E_MET_CRYO_COOLDOWN_PRESSURES
{attribute 'qualified_only'}
{attribute 'strict'}
TYPE E_MET_CRYO_COOLDOWN_PRESSURES :
(
	NONE := 0,
	VAG1,		
	VAG2,		
	VAG3,		
	VAGF,		
	VAGG,
	HPG1,
	HPG2		
);
END_TYPE

// DUTs/Enumerators/Routines/Cool_Down/E_MET_CRYO_COOLDOWN_STATE
{attribute 'qualified_only'}
{attribute 'strict'}
TYPE E_MET_CRYO_COOLDOWN_STATE :
(
	NONE := 0,				// Undefined state.
	CHECK_PRECONDITIONS,
	START_COOL_DOWN,
	START_FILLING_LN2,
	START_PTCS,
	START_TEMP_CTRL_PTC,
	KEEP_COOLING,
	STOPPING_COOL_DOWN,
	FINISHED,
	ERROR
	
);
END_TYPE

// DUTs/Enumerators/Routines/Cool_Down/E_MET_CRYO_COOLDOWN_SYS_STATE
{attribute 'qualified_only'}
{attribute 'strict'}
TYPE E_MET_CRYO_COOLDOWN_SYS_STATE :
(
	NONE := 0,
	OFF,					// Controller OFF, Valve closed
//	ACTIVE_STARTING_PUMPS,	// Controller ON,  Starting pumps
//	ACTIVE_PUMPS_RUNNING,	// Controller ON,  Pumps running
	ACTIVE_OPENING,			// Controller ON,  Valve opening
	ACTIVE_OPEN,			// Controller ON,  Valve open
	ACTIVE_CLOSING,			// Controller ON,  Valve closing
	ACTIVE_CLOSED,			// Controller ON,  Valve closed
//	ACTIVE_STOPPING_PUMPS,	// Controller ON,  Stopping pumps
	EMERGENCY,				// Controller ON,  Closing valve for safety reason
	ERROR					// Error in the system
);
END_TYPE

// DUTs/Enumerators/Routines/Cool_Down/E_MET_CRYO_COOLDOWN_VALVES
{attribute 'qualified_only'}
{attribute 'strict'}
TYPE E_MET_CRYO_COOLDOWN_VALVES :
(
	NONE := 0,
	PVV_P1,
	PVV_P2,		
	PVV_P3		
);
END_TYPE

// DUTs/Enumerators/Routines/Cool_Down/E_MET_CRYO_LN2_FILLING_STATE
{attribute 'qualified_only'}
{attribute 'strict'}
TYPE E_MET_CRYO_LN2_FILLING_STATE :
(
    NONE := 0,                                 // Undefined state

    CHECK_PRECONDITIONS,                       // Validate valves, sensors, supply

    START_LEVEL_CONTROL_SHA,                   // Begin LN2 level control at SHA (Stiff Ring)
    LEVEL_LOW_SHA,                             // LN2 reached low level at SHA

    START_LEVEL_CONTROL_SHC,                   // Begin LN2 control at SHC (Bottom Segment)
    LEVEL_LOW_SHC,                             // LN2 reached low level at SHC

    START_LEVEL_CONTROL_SHB,                   // Begin LN2 control at SHB (Middle Segment)
    FILLING,                                   // Actively filling LN2 (steady operation)

    RADIATION_SHIELDS_COLD,                    // Cryo shields have reached temperature
	
	START_PTCS,

    STOPPING_FILLING,                          // Controlled stop of LN2 flow
    FINISHED,                                  // Filling completed successfully

    ERROR                                      // Fault detected
);
END_TYPE

// DUTs/Enumerators/Routines/Re_Generation/E_MET_CRYO_RE_GENERATION_STATE
{attribute 'qualified_only'}
{attribute 'strict'}
TYPE E_MET_CRYO_RE_GENERATION_STATE :
(
	NONE := 0, 
	CHECK_PRECONDITIONS := 1, 
	START_HEATING, 
	KEEP_HEATING, 
	COOL_DOWN, 
	FINISHED, 
	ERROR
);
END_TYPE

// DUTs/Enumerators/Routines/Venting/E_MET_CRYO_VENTING_PRESSURES
{attribute 'qualified_only'}
{attribute 'strict'}
TYPE E_MET_CRYO_VENTING_PRESSURES :
(
	NONE := 0,
	VAG1,		
	VAG2,		
	VAG3,		
	VAGF,		
	VAGG,
	HPG1,
	HPG2		
);
END_TYPE

// DUTs/Enumerators/Routines/Venting/E_MET_CRYO_VENTING_STATE
{attribute 'qualified_only'}
{attribute 'strict'}
TYPE E_MET_CRYO_VENTING_STATE :
(
	NONE := 0, 
	CHECK_PRECONDITIONS := 1,
	PREPARE_FOR_VENTING,   // 2 minutes Timeout before Venting starts
	START_VENTING,
	VENTING_IN_PROGRESS,
	STOPPING_VENTING,
	FINISHED,
	ERROR
);
END_TYPE

// DUTs/Enumerators/Routines/Venting/E_MET_CRYO_VENTING_SYS_STATE
{attribute 'qualified_only'}
{attribute 'strict'}
TYPE E_MET_CRYO_VENTING_SYS_STATE :
(
	NONE := 0,
	OFF,					// Controller OFF, Valve closed
//	ACTIVE_STARTING_PUMPS,	// Controller ON,  Starting pumps
//	ACTIVE_PUMPS_RUNNING,	// Controller ON,  Pumps running
	ACTIVE_OPENING,			// Controller ON,  Valve opening
	ACTIVE_OPEN,			// Controller ON,  Valve open
	ACTIVE_CLOSING,			// Controller ON,  Valve closing
	ACTIVE_CLOSED,			// Controller ON,  Valve closed
//	ACTIVE_STOPPING_PUMPS,	// Controller ON,  Stopping pumps
	EMERGENCY,				// Controller ON,  Closing valve for safety reason
	ERROR					// Error in the system
);
END_TYPE

// DUTs/Enumerators/Routines/Venting/E_MET_CRYO_VENTING_VALVES
{attribute 'qualified_only'}
{attribute 'strict'}
TYPE E_MET_CRYO_VENTING_VALVES :
(
	NONE := 0,
	N2V_1,		
	N2V_2		
);
END_TYPE

// DUTs/Enumerators/Routines/WarmUp/E_MET_CRYO_WARMUP_STATE
{attribute 'qualified_only'}
{attribute 'strict'}
TYPE E_MET_CRYO_WARMUP_STATE :
(
	NONE := 0, 
	CHECK_PRECONDITIONS := 1, 
	START_WARM_UP,
	STOP_PTCs,
 	START_RAMP_Up_DETECTORS_1K,
	KEEP_RAMPING_Up_DETECTORS, // until detectors are at 80K
	RAMP_UP_DETECTORS_6K,
	START_RAMP_Up_RADIATION_SHIELDS,
	START_RAMP_Up_IMG,
	START_RAMP_Up_SCAO,
	START_RAMP_Up_LMS,
	START_RAMP_Up_CFO,
	KEEP_WARMING_UP, 
	STOPPING_WARM_UP,
	FINISHED, 
	ERROR
);
END_TYPE

// DUTs/Enumerators/Sensors/Base_Sensor/E_METIS_SENSOR_SOURCE
{attribute 'qualified_only'}
{attribute 'strict'}
TYPE E_METIS_SENSOR_SOURCE :
(
	NONE   := 0,
	LS240,
	LS336,
    EL32XX,
	VOTER,
	RAMP,
    DEW_POINT_CALC
);
END_TYPE

// DUTs/Enumerators/Sensors/Base_Sensor/E_METIS_SENSOR_TYPE
{attribute 'qualified_only'}
{attribute 'strict'}
TYPE E_METIS_SENSOR_TYPE :
(
	NONE        := 0,
	TEMPERATURE := 1,
	HUMIDITY    := 2
);
END_TYPE

// DUTs/Enumerators/Sensors/LN2_Level_Sensor/E_METIS_CRYO_LN2_SENSOR_LEVELS
{attribute 'qualified_only'}
{attribute 'strict'}
TYPE E_METIS_CRYO_LN2_SENSOR_LEVELS :
(
	LOW_ALARM	:= 0,	// LN2 Level is alarming low
	LOW 		:= 1,	// LN2 Level is low
	HIGH		:= 2,	// LN2 Level is High 
	HIGH_ALARM	:= 3,	// LN2 Level is alarming High
	Error		:= 4,	// Error in temperature sensors readings
	NO_LN2		:= 5    // Insufficient LN2 supply 
);
END_TYPE

// DUTs/Enumerators/Sensors/Temperature Sensor/E_METIS_LAKE_SHORE_TYPE
{attribute 'qualified_only'}
{attribute 'strict'}
TYPE E_METIS_LAKE_SHORE_TYPE :
(
	NONE 	:= 0,
	LS240	:= 1,
	LS336	:= 2,
    VOTER   := 3, // voter output
    RAMP    := 4 // ramp output
);
END_TYPE

// DUTs/Enumerators/Sensors/Temperature Sensor/E_METIS_TEMP_VOTE_METHOD
{attribute 'qualified_only'}
{attribute 'strict'}
TYPE E_METIS_TEMP_VOTE_METHOD :
(
	LOWEST_TEMPERATURE 		:= 0,
	HIGHEST_TEMPERATURE		:= 1,
	AVERAGE					:= 2,
	FIRST_VALID_TEMPERATURE	:= 3,
	MEDIAN
//	TEMPERATURE_1oo2,
//	TEMPERATURE_2oo3,
//	TEMPERATURE_3oo5
);
END_TYPE

// DUTs/Enumerators/System/E_METIS_CRYO_CTRL_CMD
{attribute 'qualified_only'}
{attribute 'strict'}
TYPE E_METIS_CRYO_CTRL_CMD :
(
	NONE	:= 0,
	COOL,
	WARM_UP,
	VENT,
	REGENERATE
);
END_TYPE

// DUTs/Enumerators/System/E_METIS_CRYO_CTRL_STATE
{attribute 'qualified_only'}
{attribute 'strict'}
TYPE E_METIS_CRYO_CTRL_STATE :
(
	
	NONE 			:= 0,
	WARM_PRESS,				// Warm & Pressurized
	PARTIAL_VACUUM,			// transitional state between Warm_Pres and Warm_Vacuum
	WARM_VACUUM,			// Warm & Vacuum
	COOLING_DOWN,			// Cooling down
	COLD,					// Cold, i.e. fully operational
	WARMING_UP,				// Warming up
	PARTIALLY_COLD,			// Cryostat is niether COLD nor WARM
	VENTING,				// Venting			
	ERROR					// Controller failure
);
END_TYPE

// DUTs/Structures/Base_Sensor/T_METIS_SENSOR_BASE_STATUS
TYPE T_METIS_SENSOR_BASE_STATUS EXTENDS T_CRYO_SENSOR_STATUS:
STRUCT
    {attribute 'TcHmiSymbol.Show'}
    sName:              STRING;
	eType:              E_METIS_SENSOR_TYPE;
	eSource:            E_METIS_SENSOR_SOURCE;    
    
    bWarning    : BOOL;
    sErrorText  : STRING;
    
    lrBaseValue : LREAL;  // the raw value expressed in the native units of the source 
	lrBaseRamp  : LREAL;  // the ramp value expressed in the native units of the source /min
END_STRUCT
END_TYPE

// DUTs/Structures/Ctrl_Valves/T_METIS_CTRL_VALVE_CFG
TYPE T_METIS_CTRL_VALVE_CFG :
STRUCT
    sDescription: 				STRING;   // User description of the controller   
    lrAutoScalePercent: 		LREAL; // scaling of the Auto value in % (range [0..100])
	lrBlowerNormalSetPoint:		LREAL;	// Air Blower setpoint for Normal Operations
	lrBlowerAlarmSetPoint:		LREAL;	// Air Blower setpoint during Alarm Conditions
END_STRUCT
END_TYPE

// DUTs/Structures/Ctrl_Valves/T_METIS_CTRL_VALVE_CTRL
TYPE T_METIS_CTRL_VALVE_CTRL:
STRUCT
    eCtrlMode:              E_METIS_CTRL_MODE;           // Auto/manual mode
	bManualEnable:          BOOL;			// Manual mode ON/OFF command (TRUE = ON, FALSE = OFF)
	lrManualSetpoint:       LREAL;	        // Manual mode output power to set (0 - 100%) [W]
    bReadConfig:			BOOL;
	bWriteConfig:			BOOL;
END_STRUCT
END_TYPE

// DUTs/Structures/Ctrl_Valves/T_METIS_CTRL_VALVE_IO_ANTI_FOG_BLOWER
TYPE T_METIS_CTRL_VALVE_IO_ANTI_FOG_BLOWER :
STRUCT
	q_bEnable				AT%Q*:		BOOL;	// Enable heater power
	q_nSetCurrent			AT%Q*:		INT;    // 4 - 20 mA valve ctrl
	i_nFlowFeedBackCurrent	AT%I*:		INT;	// 4 - 20 mA valve status feedback
	i_nFeedBackStatus				AT%I*:		UINT;	// EL3124 input status (might implement if needed)
END_STRUCT
END_TYPE

// DUTs/Structures/Ctrl_Valves/T_METIS_CTRL_VALVE_IO_IMG_CFO_PRECOOLING
TYPE T_METIS_CTRL_VALVE_IO_IMG_CFO_PRECOOLING :
STRUCT
	q_bEnable			AT%Q*:		BOOL;		// Enable heater power
	q_nSetVoltage		AT%Q*:		INT := 0;	// Adjustable PS voltage [0 - 16383 (0 - 5V)] for liner power supply to power the heater
	q_nSetCurrent		AT%Q*:		INT := 0;	// Adjustable PS current [0 - 16383 (0 - 4Amps)] for liner power supply to power the heater
	i_nActCurrent		AT%I*:		INT;		// Terminal state. Should be 8, i.e. OP.
	i_nStatus			AT%I*:		UINT;		// EL3164 input status (might implement if needed)
END_STRUCT
END_TYPE

// DUTs/Structures/Ctrl_Valves/T_METIS_CTRL_VALVE_STAT
TYPE T_METIS_CTRL_VALVE_STAT :
STRUCT
//The PLC shall monitor the health status OF the	Heaters:
//- heater open loop
//- heater short
//- heater current
//- heater power
//	in stable conditions (cold mode): the heater output shall NOT be AT 0% OR 100% in steady-state operation
//- under normal conditions, the heater output must not be set to “manual out” or “off”
//- correct selection of the range (low / medium / high)
// Any deviation from above shall trigger an alarm, warning or automated reaction, as appropriate.
	{attribute 'TcHmiSymbol.Show'}
	{attribute 'TcHmiSymbol.ReadOnly'}
	sName:				STRING;
	{attribute 'TcHmiSymbol.Show'}
	{attribute 'TcHmiSymbol.ReadOnly'}
    eCtrlMode:          E_METIS_CTRL_MODE;           // Actual Auto/manual mode

	bSimulated:			BOOL;				// Flag indicating if the value is simulated.

	lrSimFlow:			LREAL;				// Simulated Power [W]

	lrMaxFlow:			LREAL;				
	//lrMaxCurrent:			LREAL;				
	{attribute 'TcHmiSymbol.Show'}
	{attribute 'TcHmiSymbol.ReadOnly'}
	bWarning:			BOOL;
	{attribute 'TcHmiSymbol.Show'}
	{attribute 'TcHmiSymbol.ReadOnly'}
	bError:				BOOL;

	bHwWarning:			BOOL;
	{attribute 'TcHmiSymbol.Show'}
	{attribute 'TcHmiSymbol.ReadOnly'}
	bHwError:			BOOL;
	{attribute 'TcHmiSymbol.Show'}
	{attribute 'TcHmiSymbol.ReadOnly'}
	bActive:				BOOL := FALSE;

	bValveOpenLoop:	BOOL;

	bValveShort:		BOOL;
	{attribute 'TcHmiSymbol.Show'}
	{attribute 'TcHmiSymbol.ReadOnly'}
	lrActValveFlow:		LREAL;				// Calculated Power [W]
	{attribute 'TcHmiSymbol.Show'}
	{attribute 'TcHmiSymbol.ReadOnly'}
	lrActCurrent:			LREAL;				// Calculated Current [A]
	{attribute 'TcHmiSymbol.Show'}
	{attribute 'TcHmiSymbol.ReadOnly'}
	nValveState:		E_METIS_CRYO_CTRL_VALVE_STATE := E_METIS_CRYO_CTRL_VALVE_STATE.OFF;	
	{attribute 'TcHmiSymbol.Show'}
	{attribute 'TcHmiSymbol.ReadOnly'}
	sValveState:		STRING;	

	lrActDutyCycle:			LREAL;				//Actual Duty cycle at PWM module

	bActDutyCycleAvailable:	BOOL;				//Actual Duty cycle at PWM module
	{attribute 'TcHmiSymbol.Show'}
	{attribute 'TcHmiSymbol.ReadOnly'}
    lrAutoSetpointValue : LREAL;
	{attribute 'TcHmiSymbol.Show'}
	{attribute 'TcHmiSymbol.ReadOnly'}
    sAutoSetpointSource : STRING;
	{attribute 'TcHmiSymbol.Show'}
	{attribute 'TcHmiSymbol.ReadOnly'}
    lrAutoCtrlOut : LREAL;                          // controller output for AUTO mode
	{attribute 'TcHmiSymbol.Show'}
	{attribute 'TcHmiSymbol.ReadOnly'}
    lrActSetpoint : LREAL;
	{attribute 'TcHmiSymbol.Show'}
	{attribute 'TcHmiSymbol.ReadOnly'}
    bConfigured : BOOL;
    

    bAcceptCtrlMode_Auto : BOOL;

    bAcceptCtrlMode_Manual : BOOL;
	{attribute 'TcHmiSymbol.Show'}
	{attribute 'TcHmiSymbol.ReadOnly'}
    bManual : BOOL;
	{attribute 'TcHmiSymbol.Show'}
	{attribute 'TcHmiSymbol.ReadOnly'}
    bAuto : BOOL;
    
	bPowerCmdActive:	BOOL;
	{attribute 'TcHmiSymbol.ShowRecursively'}
	stAlarms:           T_CRYO_ALARMS;
	{attribute 'TcHmiSymbol.Show'}
	{attribute 'TcHmiSymbol.ReadOnly'}	
	bInputOver:			BOOL := FALSE;
	bInputUnder:		BOOL := FALSE;
	{attribute 'TcHmiSymbol.Show'}
	{attribute 'TcHmiSymbol.ReadOnly'}
	lrActFlow:			LREAL; // Actual flow percentage of opening of valve
// EL2819 Diagnostics
	{attribute 'TcHmiSymbol.Show'}
	{attribute 'TcHmiSymbol.ReadOnly'}	
	bOpenLoad        : BOOL;
	{attribute 'TcHmiSymbol.Show'}
	{attribute 'TcHmiSymbol.ReadOnly'}
	bShortTo24V      : BOOL;
	{attribute 'TcHmiSymbol.Show'}
	{attribute 'TcHmiSymbol.ReadOnly'}
	bOverCurrent     : BOOL;
	{attribute 'TcHmiSymbol.Show'}
	{attribute 'TcHmiSymbol.ReadOnly'}
	bOverTemperature : BOOL;
	{attribute 'TcHmiSymbol.Show'}
	{attribute 'TcHmiSymbol.ReadOnly'}
	bValveOpenLoadError     : BOOL;
	{attribute 'TcHmiSymbol.Show'}
	{attribute 'TcHmiSymbol.ReadOnly'}
	bValveShortCircuitError : BOOL;
	{attribute 'TcHmiSymbol.Show'}
	{attribute 'TcHmiSymbol.ReadOnly'}
	bValveFeedbackError     : BOOL;

END_STRUCT
END_TYPE

// DUTs/Structures/Error_Handeling/T_METIS_CRYO_ERROR_STATUS
TYPE T_METIS_CRYO_ERROR_STATUS :
STRUCT
    nCode      : UDINT;
    sMessage   : STRING(255);
END_STRUCT
END_TYPE

// DUTs/Structures/Heaters/METIS_HEATER/T_METIS_HEATER_CFG
TYPE T_METIS_HEATER_CFG :
STRUCT
		{attribute 'TcHmiSymbol.Show'}
    sDescription        : STRING;   // User description of the controller 
    	{attribute 'TcHmiSymbol.Show'}
    lrAutoScalePercent  : LREAL; // scaling of the Auto value in % (range [0..100])
    
END_STRUCT
END_TYPE

// DUTs/Structures/Heaters/METIS_HEATER/T_METIS_HEATER_CTRL
TYPE T_METIS_HEATER_CTRL:
STRUCT
		{attribute 'TcHmiSymbol.Show'}
    eCtrlMode:              E_METIS_CTRL_MODE;           // Auto/manual mode
		{attribute 'TcHmiSymbol.Show'}
	bManualEnable:          BOOL;			// Manual mode ON/OFF command (TRUE = ON, FALSE = OFF)
		{attribute 'TcHmiSymbol.Show'}
	lrManualSetpoint:       LREAL;	        // Manual mode output power to set (0 - 100%) [W]
		{attribute 'TcHmiSymbol.Show'}
    bReadConfig:			BOOL;
		{attribute 'TcHmiSymbol.Show'}
	bWriteConfig:			BOOL;
END_STRUCT
END_TYPE

// DUTs/Structures/Heaters/METIS_HEATER/T_METIS_HEATER_IO_CPAU60
TYPE T_METIS_HEATER_IO_CPAU60 :
STRUCT
	q_bEnable			AT%Q*:		BOOL;	// Enable heater power
	q_nSetVoltage		AT%Q*:		INT;    // Adjustable PS voltage [0 - 16383 (0 - 5V)] for liner power supply to power the heater
	i_nActCurrent		AT%I*:		DINT;	// Terminal state. Should be 8, i.e. OP.
	i_nStatus			AT%I*:		UINT;	// EL3164 input status (might implement if needed)
END_STRUCT
END_TYPE

// DUTs/Structures/Heaters/METIS_HEATER/T_METIS_HEATER_IO_CXWUI60
TYPE T_METIS_HEATER_IO_CXWUI60 :
STRUCT
	q_bEnable			AT%Q*:		BOOL;		// Enable heater power
	q_nSetVoltage		AT%Q*:		INT := 0;	// Adjustable PS voltage [0 - 16383 (0 - 5V)] for liner power supply to power the heater
	q_nSetCurrent		AT%Q*:		INT := 0;	// Adjustable PS current [0 - 16383 (0 - 4Amps)] for liner power supply to power the heater
	i_nActCurrent		AT%I*:		INT;		// Terminal state. Should be 8, i.e. OP.
	i_nStatus			AT%I*:		UINT;		// EL3164 input status (might implement if needed)
END_STRUCT
END_TYPE

// DUTs/Structures/Heaters/METIS_HEATER/T_METIS_HEATER_IO_EL95X1
TYPE T_METIS_HEATER_IO_EL95X1 :
STRUCT
	i_bOutputOverload   AT %I*:	BOOL; // AO Output Status - Output Overload
	i_bUnderrange       AT %I*:	BOOL; // AO Output Status - Underrange
	i_bOverrange        AT %I*:	BOOL; // AO Output Status - Overrange
	i_bWarning 			AT %I*: BOOL; // AO Output Status - Warning
	i_bError			AT %I*: BOOL; // AO Output Status - Error
    
    i_rVoltage          AT %I*: REAL; // 0x1A53 (AI Output Voltage Compact Real32) - Value (Real32)
    i_rCurrent          AT %I*: REAL; // 0x1A63 (AI Output Current Compact Real32) - Value (Real32)
    
    q_bEnable			AT %Q*:	BOOL;   // Enable heater power via relay
    q_rSetVoltage       AT %Q*: REAL;   // EL95X1 - AO Output Standard (Real32) - Value
    q_nOutputInterface  AT %Q*: UINT;   // EL95X1 - AO Output Standard (Real32) - Control - Output interface
    q_nOutputOperation  AT %Q*: UINT;   // EL95X1 - AO Output Standard (Real32) - Control - Output operation 
END_STRUCT
END_TYPE

// DUTs/Structures/Heaters/METIS_HEATER/T_METIS_HEATER_IO_PWM
TYPE T_METIS_HEATER_IO_PWM :
STRUCT
	i_nActCurrent		AT %I*:	INT;    // Terminal state. Should be 8, i.e. OP.
	i_bReadyToEnable 	AT %I*:	BOOL;
	i_bWarning 			AT %I*: BOOL;
	i_bError			AT %I*: BOOL;
	i_nDuty_Cycle		AT %I*: INT;
	q_bEnable			AT %Q*:	BOOL;   // Enable heater power
	q_bEnableDithering	AT %Q*: BOOL;
	q_bReset			AT %Q*: BOOL;
	q_nPWMOut			AT %Q*: INT;	// 
END_STRUCT
END_TYPE

// DUTs/Structures/Heaters/METIS_HEATER/T_METIS_HEATER_STAT
TYPE T_METIS_HEATER_STAT :
STRUCT
//The PLC shall monitor the health status OF the	Heaters:
//- heater open loop
//- heater short
//- heater current
//- heater power
//	in stable conditions (cold mode): the heater output shall NOT be AT 0% OR 100% in steady-state operation
//- under normal conditions, the heater output must not be set to “manual out” or “off”
//- correct selection of the range (low / medium / high)
// Any deviation from above shall trigger an alarm, warning or automated reaction, as appropriate.
	{attribute 'TcHmiSymbol.Show'}
	{attribute 'TcHmiSymbol.ReadOnly'}
	sName:				STRING;
	{attribute 'TcHmiSymbol.Show'}
	{attribute 'TcHmiSymbol.ReadOnly'}
    eCtrlMode:          E_METIS_CTRL_MODE;           // Actual Auto/manual mode
	{attribute 'TcHmiSymbol.Show'}
	{attribute 'TcHmiSymbol.ReadOnly'}
	bSimulated:			BOOL;				// Flag indicating if the value is simulated.
	{attribute 'TcHmiSymbol.Show'}
	{attribute 'TcHmiSymbol.ReadOnly'}
	lrSimPower:			LREAL;				// Simulated Power [W]
	{attribute 'TcHmiSymbol.Show'}
	{attribute 'TcHmiSymbol.ReadOnly'}
	lrMaxPower:			LREAL;				
	{attribute 'TcHmiSymbol.Show'}
	{attribute 'TcHmiSymbol.ReadOnly'}
	lrMaxCurrent:			LREAL;				
	{attribute 'TcHmiSymbol.Show'}
	{attribute 'TcHmiSymbol.ReadOnly'}
	bWarning:			BOOL;
	{attribute 'TcHmiSymbol.Show'}
	{attribute 'TcHmiSymbol.ReadOnly'}
	bError:				BOOL;
	{attribute 'TcHmiSymbol.Show'}
	{attribute 'TcHmiSymbol.ReadOnly'}
	bHwWarning:			BOOL;
	{attribute 'TcHmiSymbol.Show'}
	{attribute 'TcHmiSymbol.ReadOnly'}
	bHwError:			BOOL;
	{attribute 'TcHmiSymbol.Show'}
	{attribute 'TcHmiSymbol.ReadOnly'}
	bActive:				BOOL := FALSE;
	{attribute 'TcHmiSymbol.Show'}
	{attribute 'TcHmiSymbol.ReadOnly'}
	bHeaterOpenLoop:	BOOL;
	{attribute 'TcHmiSymbol.Show'}
	{attribute 'TcHmiSymbol.ReadOnly'}
	bHeaterShort:		BOOL;
	{attribute 'TcHmiSymbol.Show'}
	{attribute 'TcHmiSymbol.ReadOnly'}
	lrActHeaterPower:		LREAL;				// Calculated Power [W]
	{attribute 'TcHmiSymbol.Show'}
	{attribute 'TcHmiSymbol.ReadOnly'}
	lrActCurrent:			LREAL;				// Calculated Current [A]
	{attribute 'TcHmiSymbol.Show'}
	{attribute 'TcHmiSymbol.ReadOnly'}
	lrActVoltage: LREAL;                        // Measured voltage [V] (e.g. for EL9501/EL9561)
	{attribute 'TcHmiSymbol.Show'}
	{attribute 'TcHmiSymbol.ReadOnly'}
	nHeaterState:		E_METIS_CRYO_HEATER_STATE := E_METIS_CRYO_HEATER_STATE.OFF;	
	{attribute 'TcHmiSymbol.Show'}
	{attribute 'TcHmiSymbol.ReadOnly'}
	sHeaterState:		STRING;	
	{attribute 'TcHmiSymbol.Show'}
	{attribute 'TcHmiSymbol.ReadOnly'}
	lrActDutyCycle:			LREAL;				//Actual Duty cycle at PWM module
    {attribute 'TcHmiSymbol.Show'}
	{attribute 'TcHmiSymbol.ReadOnly'}
	bActDutyCycleAvailable:	BOOL;				//Actual Duty cycle at PWM module
	{attribute 'TcHmiSymbol.Show'}
	{attribute 'TcHmiSymbol.ReadOnly'}
    lrAutoSetpointValue : LREAL;
	{attribute 'TcHmiSymbol.Show'}
	{attribute 'TcHmiSymbol.ReadOnly'}
    sAutoSetpointSource : STRING;
	{attribute 'TcHmiSymbol.Show'}
	{attribute 'TcHmiSymbol.ReadOnly'}
    lrAutoCtrlOut : LREAL;                          // controller output for AUTO mode
	{attribute 'TcHmiSymbol.Show'}
	{attribute 'TcHmiSymbol.ReadOnly'}
    lrActSetpoint : LREAL;
	{attribute 'TcHmiSymbol.Show'}
	{attribute 'TcHmiSymbol.ReadOnly'}
    bConfigured : BOOL;
    
	{attribute 'TcHmiSymbol.Show'}
	{attribute 'TcHmiSymbol.ReadOnly'}
    bAcceptCtrlMode_Auto : BOOL;
	{attribute 'TcHmiSymbol.Show'}
	{attribute 'TcHmiSymbol.ReadOnly'}
    bAcceptCtrlMode_Manual : BOOL;
	{attribute 'TcHmiSymbol.Show'}
	{attribute 'TcHmiSymbol.ReadOnly'}
    bManual : BOOL;
	{attribute 'TcHmiSymbol.Show'}
	{attribute 'TcHmiSymbol.ReadOnly'}
    bAuto : BOOL;
	{attribute 'TcHmiSymbol.Show'}
	{attribute 'TcHmiSymbol.ReadOnly'}
	bHeaterThermalSwitchOpen : BOOL;
	{attribute 'TcHmiSymbol.Show'}
	{attribute 'TcHmiSymbol.ReadOnly'}
	bHeaterInsufficientPower : BOOL;
	{attribute 'TcHmiSymbol.Show'}
	{attribute 'TcHmiSymbol.ReadOnly'}
	lrExpectedHeaterPower    : LREAL;
	{attribute 'TcHmiSymbol.Show'}
	{attribute 'TcHmiSymbol.ReadOnly'}
	lrHeaterPowerRatio       : LREAL;
	
    
	bPowerCmdActive:	BOOL;
	{attribute 'TcHmiSymbol.ShowRecursively'}
	stAlarms:           T_CRYO_ALARMS;

END_STRUCT
END_TYPE

// DUTs/Structures/Heaters/T_METIS_CRYO_HEATER_CTRL
TYPE T_METIS_CRYO_HEATER_CTRL:
STRUCT
	bEnable:	BOOL;			// Control to Start/Stop the heater.
	bPower:		BOOL;			// Update heater power output.
	lrPower:	LREAL:= 0.0;	// Output power to set (0 - 100%) [W] 
END_STRUCT
END_TYPE

// DUTs/Structures/Heaters/T_METIS_CRYO_HEATER_STATUS
TYPE T_METIS_CRYO_HEATER_STATUS :
STRUCT
//The PLC shall monitor the health status OF the	Heaters:
//- heater open loop
//- heater short
//- heater current
//- heater power
//	in stable conditions (cold mode): the heater output shall NOT be AT 0% OR 100% in steady-state operation
//- under normal conditions, the heater output must not be set to “manual out” or “off”
//- correct selection of the range (low / medium / high)
// Any deviation from above shall trigger an alarm, warning or automated reaction, as appropriate.
	{attribute 'TcHmiSymbol.Show'}
	{attribute 'TcHmiSymbol.ReadOnly'}
	sName:				STRING;
	{attribute 'TcHmiSymbol.Show'}
	{attribute 'TcHmiSymbol.ReadOnly'}
	bSimulated:			BOOL;				// Flag indicating if the value is simulated.
	{attribute 'TcHmiSymbol.Show'}
	{attribute 'TcHmiSymbol.ReadOnly'}
	lrSimPower:			LREAL;				// Simulated Power [W]
	{attribute 'TcHmiSymbol.Show'}
	{attribute 'TcHmiSymbol.ReadOnly'}
	lrMaxPower:			LREAL;				
	{attribute 'TcHmiSymbol.Show'}
	{attribute 'TcHmiSymbol.ReadOnly'}
	lrMaxCurrent:			LREAL;				
	{attribute 'TcHmiSymbol.Show'}
	{attribute 'TcHmiSymbol.ReadOnly'}
	bWarning:			BOOL;
	{attribute 'TcHmiSymbol.Show'}
	{attribute 'TcHmiSymbol.ReadOnly'}
	bError:				BOOL;
	{attribute 'TcHmiSymbol.Show'}
	{attribute 'TcHmiSymbol.ReadOnly'}
	bHwWarning:			BOOL;
	{attribute 'TcHmiSymbol.Show'}
	{attribute 'TcHmiSymbol.ReadOnly'}
	bHwError:			BOOL;
	{attribute 'TcHmiSymbol.Show'}
	{attribute 'TcHmiSymbol.ReadOnly'}
	bActive:				BOOL := FALSE;
	{attribute 'TcHmiSymbol.Show'}
	{attribute 'TcHmiSymbol.ReadOnly'}
	bHeaterOpenLoop:	BOOL;
	{attribute 'TcHmiSymbol.Show'}
	{attribute 'TcHmiSymbol.ReadOnly'}
	bHeaterShort:		BOOL;
	{attribute 'TcHmiSymbol.Show'}
	{attribute 'TcHmiSymbol.ReadOnly'}
	lrActHeaterPower:		LREAL;				// Calculated Power [W]
	{attribute 'TcHmiSymbol.Show'}
	{attribute 'TcHmiSymbol.ReadOnly'}
	lrActCurrent:			LREAL;				// Calculated Current [A]
	{attribute 'TcHmiSymbol.Show'}
	{attribute 'TcHmiSymbol.ReadOnly'}
	nHeaterState:		E_METIS_CRYO_HEATER_STATE := E_METIS_CRYO_HEATER_STATE.OFF;	
	{attribute 'TcHmiSymbol.Show'}
	{attribute 'TcHmiSymbol.ReadOnly'}
	sHeaterState:		STRING;	
	{attribute 'TcHmiSymbol.Show'}
	{attribute 'TcHmiSymbol.ReadOnly'}
	lrActDutyCycle:			LREAL;				//Actual Duty cycle at PWM modile
	
	bPowerCmdActive:	BOOL;
	stAlarms:           T_CRYO_ALARMS;

END_STRUCT
END_TYPE

// DUTs/Structures/LN2_Level_Ctrl/T_LN2_LEVEL_CTRL_CFG
TYPE T_LN2_LEVEL_CTRL_CFG :
STRUCT
	{attribute 'TcHmiSymbol.Show'}
	lrLN2_Level_SenseTempK_HA:		LREAL := 90.0; // Threshold temperature read by the heated pt100s when submerged under LN2
	{attribute 'TcHmiSymbol.Show'}
	lrLN2_Level_SenseTempK_H:		LREAL := 85.0;
	{attribute 'TcHmiSymbol.Show'}
	lrLN2_Level_SenseTempK_L:		LREAL := 85.0;
	{attribute 'TcHmiSymbol.Show'}
	lrLN2_Level_SenseTempK_LA:		LREAL := 85.0;
	{attribute 'TcHmiSymbol.Show'}	
	lrLN2_Level_AbsenceTempK_HA:	LREAL := 90.0; 	// Threshold temperature read by the heated pt100s when LN2 is absent OR Evaporated 
	{attribute 'TcHmiSymbol.Show'}
	lrLN2_Level_AbsenceTempK_H:		LREAL := 85.0;
	{attribute 'TcHmiSymbol.Show'}
	lrLN2_Level_AbsenceTempK_L:		LREAL := 85.0;
	{attribute 'TcHmiSymbol.Show'}
	lrLN2_Level_AbsenceTempK_LA:	LREAL := 85.0;
	{attribute 'TcHmiSymbol.Show'}
	lr_Early_Refill_Duration_Time: 	LREAL := 24.0; // When Cooldown starts, LN2 level control not wait for the LOW sensor before starting the refilling
	{attribute 'TcHmiSymbol.Show'}
	lr_Cycle_Time: 					LREAL := 2.0; // During Early refill, Refilling will restart after tCycle_Time
	{attribute 'TcHmiSymbol.Show'}
	lr_LN2Level_Hold_Time:			LREAL := 20.0; 	// LN2 level change hold time for 
END_STRUCT
END_TYPE

// DUTs/Structures/LN2_Level_Ctrl/T_LN2_LEVEL_CTRL_CTRL
TYPE T_LN2_LEVEL_CTRL_CTRL :
STRUCT
		{attribute 'TcHmiSymbol.Show'}
    bReadConfig:			BOOL;
		{attribute 'TcHmiSymbol.Show'}
	bWriteConfig:			BOOL;
END_STRUCT
END_TYPE

// DUTs/Structures/PID_Control/Generic/E_METIS_CTRL_MODE
{attribute 'qualified_only'}
{attribute 'strict'}
TYPE E_METIS_CTRL_MODE :
(
	NONE := 0,
    AUTO := 1,
    MANUAL := 2
);
END_TYPE

// DUTs/Structures/PID_Control/Generic/E_METIS_CTRL_SETPOINT_SWITCH
{attribute 'qualified_only'}
{attribute 'strict'}
TYPE E_METIS_CTRL_SETPOINT_SWITCH :
(
	FIXED := 0,
    VARIABLE
);
END_TYPE

// DUTs/Structures/PID_Control/Generic/T_METIS_CTRL_LOOP_CFG
{attribute 'TcHmiSymbol.ShowRecursively'}
TYPE T_METIS_CTRL_LOOP_CFG:
STRUCT
    // general
    bEnabled            : BOOL;             // TRUE to enable the control loop automatically   
    sDescription        : STRING;   // User description of the controller 
    
    sInputTempName      : STRING;
    sSetpointTempName   : STRING;
    
    eSetpointSwitch     : E_METIS_CTRL_SETPOINT_SWITCH;
    
    lrFixedSetpoint     : LREAL;
    lrSetpointOffset    : LREAL;
	lrManualOut		: LREAL		:= 0.0;
        
    bSyncManualOut : BOOL; // sync manual output value to auto output value
    
    
	// Ramp
	lrRampUpRate        : LREAL		:= 60;	// Ramp up rate in units per second 
	lrRampDownRate      : LREAL		:= 60;	// Ramp down rate in units per second
    
	// PID Parameters
	lrKp                : LREAL := 1.0;     // Controller amplification / controller coefficient
  	lrTn                : LREAL := 0.0; 	// Integral action time in seconds; if this is parameterized to 0s, the I component is deactivated.
  	lrTv                : LREAL := 0.0; 	// Derivative action time in seconds; if this is parameterized to 0s, the D component is deactivated.
	lrTd                : LREAL := 0.0;     // Damping time in seconds
    
    
    eStartupCtrlMode       : E_METIS_CTRL_MODE;    // AUTO or MANUAL
    nStartupTimeout        : DINT  := 5000;        // startup timeout in [ms] during which the inputs must become valid
                                                  // (otherwise the output switches to MANUAL)
                                                  
    nInputTempTimeout      : DINT := 60000;    // the control loop will only switch to MANUAL if the input temperature becomes invalid for more than this time
    nSetpointTempTimeout   : DINT := 60000;    // the control loop will only switch to MANUAL if the setpoint temperature becomes invalid for more than this time

END_STRUCT
END_TYPE

// DUTs/Structures/PID_Control/Generic/T_METIS_CTRL_LOOP_CTRL
{attribute 'TcHmiSymbol.ShowRecursively'}
TYPE T_METIS_CTRL_LOOP_CTRL:
STRUCT
    // general
    
    eCtrlMode:      E_METIS_CTRL_MODE;  // AUTO or MANUAL
    bEngMode:       BOOL;   // TRUE means engineering mode should be ON
    
    bHold   : BOOL; // level-based
    
    lrFixedSetpoint : LREAL;
    lrSetpointOffset : LREAL;
    
    // 	
	//lrRampSetpointValue		: LREAL		:= 0.0;
	lrManualOut		: LREAL		:= 0.0;
    
    nInputTempIndex : INT;
    nSetpointTempIndex : INT;
    
    // config reading/writing
	bReadConfig         : BOOL;     // start reading the config file
	bWriteConfig        : BOOL;     // start writing the config file
    
    // output
    lrOutMaxLimit       : LREAL := 100.0;
    lrOutMinLimit       : LREAL := 0.0;
    
    // clear some diagnostics
    bClearForcedManualDiag : BOOL;
	
	eInputTempIndex:		 	E_ALL_METIS_TEMPERATURES;
	eVariableSetpointIndex:		E_ALL_METIS_TEMPERATURES;
END_STRUCT
END_TYPE

// DUTs/Structures/PID_Control/Generic/T_METIS_CTRL_LOOP_STAT
{attribute 'TcHmiSymbol.ShowRecursively'}
TYPE T_METIS_CTRL_LOOP_STAT:
STRUCT
	bConfigured:	BOOL	:= FALSE;
	bDone:			BOOL;			// Flag if controller is OK
	bBusy:			BOOL;			// Flag if controller is BUSY
	bError:			BOOL;			// Flag if controller is in ERROR state
	bValid:         BOOL;			// Flag if controller is OK
    bStarted:       BOOL;
    
    eCtrlMode:      E_METIS_CTRL_MODE;  // AUTO or MANUAL
    bEngMode:       BOOL; 
    
    bAcceptCtrlMode_Auto     : BOOL;
    bAcceptCtrlMode_Manual   : BOOL;
    
    
	nCycleCounter:	UDINT := 0;
	nState:			E_CRYO_BIN_CTRL_STATE	:= E_CRYO_BIN_CTRL_STATE.NONE;

	sState:			STRING(64);		// State as text
	sError:			STRING(64);		// Error as text
	
	
	bInterlock:	BOOL := FALSE;	// Flag if any command is prevented
	bWarning:	BOOL := FALSE;	// ENG command set to a not permitted command
	sMode:		STRING := '';	// Active Mode
	sStatus:	STRING := 'OK';	// Textual description in case of problems

	// ON/OFF command permissions
	bPermitOn:		BOOL := TRUE;
	bPermitOff:		BOOL := TRUE;
    
    lrTargetSetpoint   : LREAL;
    lrActInput      : LREAL;
    sActInputDescription : STRING;
    bActInputValid : BOOL;
    lrActVariableSetpoint : LREAL;
    bActVariableSetpointValid : BOOL;
    lrRampValue     : LREAL;
    sActVariableSetpointDescription : STRING;
    
    bARWactive : BOOL;
    nErrorId : INT;
    
    lrControllerOut : LREAL;
    
    // some redundant helper variables (for simplifying HMI development)
    bSetpointSwitchIsFixed : BOOL;
    bSetpointSwitchIsVariable : BOOL;
    bCtrlModeIsAuto : BOOL;
    bCtrlModeIsManual : BOOL;
    
    // extra diagnostics
    sLastForcedManualTime : STRING;
    sLastForcedManualCause : STRING;
	{attribute 'TcHmiSymbol.ShowRecursively'}
	{attribute 'TcHmiSymbol.ReadOnly'}
	stAlarms:		T_CRYO_ALARMS;	

END_STRUCT
END_TYPE

// DUTs/Structures/PID_Control/T_METIS_CTRL_BASE_CFG
TYPE T_METIS_CTRL_BASE_CFG :
STRUCT
	(* Ramp *)
	lrRampUpRate			: LREAL		:= 60;	(* in units per second *) 
	lrRampDownRate		  	: LREAL		:= 60;	(* in units per second *)
	(*PID Parameters*)
	lrKp                    : LREAL := 1; 		// Controller amplification / controller coefficient
  	tTn                    	: TIME := T#0MS; 	// Integral action time; if this is parameterized to T#0s, the I component is deactivated.
  	tTv                    	: TIME := T#0MS; 	// Derivative action time; if this is parameterized to T#0s, the D component is deactivated.
	tTd					   	: TIME := T#0MS;
END_STRUCT
END_TYPE

// DUTs/Structures/PID_Control/T_METIS_CTRL_BASE_CTRL
TYPE T_METIS_CTRL_BASE_CTRL :
STRUCT
	(* input *)
	bEnable									: BOOL		:= FALSE;	
	lrRampSetpointValue						: LREAL		:= 273.0;
	lrManualSetPoint						: LREAL		:= 273.0;
	lrManualRampUpRate						: LREAL		:= 2;
	lrManualRampDownRate					: LREAL		:= 2;
END_STRUCT
END_TYPE

// DUTs/Structures/PID_Control/T_METIS_CTRL_BASE_STAT
TYPE T_METIS_CTRL_BASE_STAT :
STRUCT
	bEnabled:		BOOL 	:= FALSE;	// Controller active while bEnable is TRUE
	bConfigured:	BOOL	:= FALSE;
	bDone:			BOOL;			// Flag if controller is OK
	bBusy:			BOOL;			// Flag if controller is BUSY
	bError:			BOOL;			// Flag if controller is in ERROR state
	bActive:		BOOL;			// Flag if controller is ACTIVE

	nCycleCounter:	UDINT := 0;
	nState:			E_CRYO_BIN_CTRL_STATE	:= E_CRYO_BIN_CTRL_STATE.NONE;

	sState:			STRING(64);		// State as text
	sError:			STRING(64);		// Error as text
	
	
	bInterlock:	BOOL := FALSE;	// Flag if any command is prevented
	bWarning:	BOOL := FALSE;	// ENG command set to a not permitted command
	sMode:		STRING := '';	// Active Mode
	sStatus:	STRING := 'OK';	// Textual description in case of problems

	// ON/OFF command permissions
	bPermitOn:		BOOL := TRUE;
	bPermitOff:		BOOL := TRUE;
END_STRUCT
END_TYPE

// DUTs/Structures/RAMP/T_METIS_CTRL_RAMP_CTRL
TYPE T_METIS_CTRL_RAMP_CTRL :
STRUCT
	(* input *)
	bEnable											: BOOL		:= FALSE;
	fStart											: LREAL 	:= 0.0;
	fTarget											: LREAL		:= 5.0;
	
	bInit											: BOOL 		:= FALSE; (* To initialize the required ramp*)
	
	(* Ramp *)
	RampUp_Rate										: LREAL		:= 60;	(* in units per second *) 
	RampDown_Rate									: LREAL		:= 60;	(* in units per second *)
END_STRUCT
END_TYPE

// DUTs/Structures/RAMP/T_METIS_CTRL_RAMP_STAT
TYPE T_METIS_CTRL_RAMP_STAT :
STRUCT
	
	fOut				: LREAL;		
    bValueReached		: BOOL;
    bError				: BOOL;
    eErrorId			: E_CTRL_ERRORCODES;
	bConfigured			: BOOL;
	
END_STRUCT
END_TYPE

// DUTs/Structures/Routines/Anti_Fogging/T_MET_CRYO_ANTI_FOGGING_CTRL
TYPE T_MET_CRYO_ANTI_FOGGING_CTRL :
STRUCT

	bEnable:						BOOL := FALSE;
	bStop:							BOOL := FALSE;
	bReset:							BOOL := FALSE;
END_STRUCT
END_TYPE

// DUTs/Structures/Routines/Anti_Fogging/T_MET_CRYO_ANTI_FOGGING_STAT
TYPE T_MET_CRYO_ANTI_FOGGING_STAT :
STRUCT
	

	bEnabled:				BOOL := FALSE;	// Controller active while bEnable is TRUE
	bConfigured:			BOOL := FALSE;	// Flag if controller has been configured.
	bError:					BOOL;			// Flag if controller is OK
	bActive:				BOOL:= FALSE;			// Flag if controller is ACTIVE
	bDone:					BOOL;			// Flag if controller is OK
	bBusy:					BOOL;			// Flag if controller is BUSY
	bAlarm:					BOOL := FALSE;
	bWarning:				BOOL := FALSE;
	
	bEmergency:				BOOL := FALSE;	// Flag if there was Emergency valve closure
	bPreConditionsMet:		BOOL := FALSE;
	bAuto:					BOOL := TRUE;

	nState:					E_MET_CRYO_ANTI_FOGGING_STATE	:= E_MET_CRYO_ANTI_FOGGING_STATE.NONE;
	nAntiFoggingMode:		E_ANTI_FOGGING_MODE := E_ANTI_FOGGING_MODE.PURGING;			
	
	
	
	
	sState:			STRING(64);		// State as text
	sStatus:		STRING(64);		// Status as text
	sErrorText:		STRING(64);		// Error as text
	
	bPermitEvacuationStop:			BOOL := TRUE;
	bPermitVenting:					BOOL := TRUE;
	
	// Error handeling	

	Error: 		T_METIS_CRYO_ERROR_STATUS;
	sErrorMessage:		STRING(256) := '';		// Error message	
	nErrorCode:			UDINT := 0;
	sRecoverySuggestion: STRING(256) := '';
	

END_STRUCT
END_TYPE

// DUTs/Structures/Routines/Cool_Down/T_MET_CRYO_COOLDOWN_CFG
TYPE T_MET_CRYO_COOLDOWN_CFG :
STRUCT
	// Pressure sensor gauge types
	nType_VAG1:		E_CRYO_SENSOR_TYPE_PRESS := E_CRYO_SENSOR_TYPE_PRESS.PKR_360;
	nType_VAG2:		E_CRYO_SENSOR_TYPE_PRESS := E_CRYO_SENSOR_TYPE_PRESS.PKR_360;
	nType_VAG3:		E_CRYO_SENSOR_TYPE_PRESS := E_CRYO_SENSOR_TYPE_PRESS.PKR_360;
	nType_VAGF1:	E_CRYO_SENSOR_TYPE_PRESS := E_CRYO_SENSOR_TYPE_PRESS.PKR_360;
	nType_VAGF2:	E_CRYO_SENSOR_TYPE_PRESS := E_CRYO_SENSOR_TYPE_PRESS.PKR_360;
	nType_VAGG1:	E_CRYO_SENSOR_TYPE_PRESS := E_CRYO_SENSOR_TYPE_PRESS.PKR_360;
	nType_VAGG2:	E_CRYO_SENSOR_TYPE_PRESS := E_CRYO_SENSOR_TYPE_PRESS.PKR_360;
	nType_HPG1:		E_CRYO_SENSOR_TYPE_PRESS := E_CRYO_SENSOR_TYPE_PRESS.CMR_361;
	nType_HPG2:		E_CRYO_SENSOR_TYPE_PRESS := E_CRYO_SENSOR_TYPE_PRESS.CMR_361;
	
	nPressGaugeType1:	E_CRYO_SENSOR_TYPE_PRESS := E_CRYO_SENSOR_TYPE_PRESS.PKR_360;
	nPressGaugeType2:	E_CRYO_SENSOR_TYPE_PRESS := E_CRYO_SENSOR_TYPE_PRESS.PKR_360;

	//bPressSimulation:	BOOL := FALSE;	// Flag is pre-vacuum pressure is simulated.

	// Flag is pressures are simulated.
	// TODO: Define individual flags for each sensor.
	//bPressSimulation:	BOOL := FALSE;	

	lrThld_Prevac:			LREAL := 0.1;	// Prevacuum pressure threshold [mbar] 
	lrThld_PrevacHigh:		LREAL := 5.0;	// Prevacuum pressure too high threshold [mbar]
	lrThld_Vacuum:			LREAL := 0.0001;// At this Cryo pressure evacuation has started [mbar]
	
	// Cryo pressure threshold for safe Turbo Pump start
	lrThld_TP_SafeStartPressure:	LREAL := 0.01;	
	// Cryo pressure threshold for safe Valve opening
	lrThld_Valve_SafeOpenPressure:	LREAL := 0.1;	
	
	tDelay:		TIME := T#3S;	// Time delay before stopping Turbo Pump
END_STRUCT
END_TYPE

// DUTs/Structures/Routines/Cool_Down/T_MET_CRYO_COOLDOWN_CTRL
TYPE T_MET_CRYO_COOLDOWN_CTRL :
STRUCT
	
	bEnable:						BOOL := FALSE;
	bStop:							BOOL := FALSE;
	bReset:							BOOL := FALSE;

	bEnable_PVV_P1:	BOOL := FALSE;
	bEnable_PVV_P2:	BOOL := FALSE;
	bEnable_PVV_P3:	BOOL := FALSE;
	

	// Override flags
	//
	
	// Valve command override handling
	cor_PVV_P1:	FB_CRYO_CMD_OVERRIDE;
	cor_PVV_P2:	FB_CRYO_CMD_OVERRIDE;
	cor_PVV_P3:	FB_CRYO_CMD_OVERRIDE;
	
	por_VAG_PCA:	FB_CRYO_CMD_OVERRIDE;
	por_VAG_PCB:	FB_CRYO_CMD_OVERRIDE;
	por_VAG_P1:		FB_CRYO_CMD_OVERRIDE;
	
	bSim_Press_VAG_PCA: 	BOOL;
	bSim_Press_VAG_PCB: 	BOOL;
	bSim_Press_VAG_P1: 		BOOL;	

	
	
	///////////////////////
	///// PTC Coolers /////
	//////////////////////	
	
	// Command override (cor)
	cor_PTC_1:				FB_CRYO_CMD_OVERRIDE;
	cor_PTC_2:				FB_CRYO_CMD_OVERRIDE;
	cor_PTC_3:				FB_CRYO_CMD_OVERRIDE;
	
	bPTC_1_Enable:		BOOL := FALSE;
	bPTC_2_Enable:		BOOL := FALSE;
	bPTC_3_Enable:		BOOL := FALSE;
	
	////////////////////////////////
	// LN2 Level Sensors & Control//
	////////////////////////////////
	cor_LN2_V1:				FB_CRYO_CMD_OVERRIDE;
	cor_LN2_V2:				FB_CRYO_CMD_OVERRIDE;
	cor_LN2_V3:				FB_CRYO_CMD_OVERRIDE;
	
	bEnable_LN2_Level_Control: ARRAY [1..3] OF BOOL;
	
	
END_STRUCT
END_TYPE

// DUTs/Structures/Routines/Cool_Down/T_MET_CRYO_COOLDOWN_STAT
TYPE T_MET_CRYO_COOLDOWN_STAT :
STRUCT
	bEnabled:		BOOL := FALSE;	// Controller active while bEnable is TRUE
	bConfigured:	BOOL := FALSE;	// Flag if controller has been configured.
	bError:			BOOL;			// Flag if controller is OK
	bActive:		BOOL;			// Flag if controller is ACTIVE
	bEmergency:		BOOL := FALSE;	// Flag if there was Emergency valve closure
	bAlarm:			BOOL := FALSE;
	bWarning:		BOOL := FALSE;
	bBusy:			BOOL := FALSE;
	bDone:			BOOL := FALSE;
	bPreConditionsMet:		BOOL := FALSE;
	//bRootPumpON:	BOOL;			// Flag if Root Pump is running
	//bTurboPumpON:	BOOL;			// Flag if Turbo Pump is running
	bPVVP1Open:		BOOL;			// Flag if venting PVV_P1 valve is open
	bPVVP2Open:		BOOL;			// Flag if venting PVV_P2 valve is open
	bPVVP3Open:		BOOL;			// Flag if venting PVV_P3 valve is open
//	bN2C2Open:		BOOL;			// Flag if venting N2C_1 valve is open
//	bVentingValvesOpen:		BOOL;	// Flag if all venting valves are open
//	bValveAfterTP:	BOOL := FALSE;	// Flag if Evacuation Valve should open after TP has started

	// Generic controller OK flag.
	// Used for problems other than from the actuator.
	// This flag is used for problems coming from controllers
	// that extend the functionality of FB_CRYO_BIN_CTRL.
	bCtrlOK:	BOOL := TRUE;		

	nCycleCounter:	UDINT := 0;
	nState:			E_MET_CRYO_COOLDOWN_STATE	:= E_MET_CRYO_COOLDOWN_STATE.NONE;
	

	sState:						STRING(80);		// State as text
	sSubState:					STRING(80);		// State as text
	
	sEarlyFillState:			STRING(80);		// State as text
	sEarlyFillSubState: 		STRING(80);		// State as text
	
	sStatus:					STRING(80);		// Status as text
	
	bPermitEvacuationStop:			BOOL := TRUE;
	
	bReadyForOperations:		BOOL := FALSE;

// Error handeling	

	Error: 		T_METIS_CRYO_ERROR_STATUS;
	sErrorMessage:		STRING(256) := '';		// Error message	
	nErrorCode:			UDINT := 0;
	sRecoverySuggestion: STRING(256) := '';
	
	
	
	nFillingState: 					E_MET_CRYO_LN2_FILLING_STATE := E_MET_CRYO_LN2_FILLING_STATE.NONE; // Used in the state-machine
	nStandAloneFillingState: 		E_MET_CRYO_LN2_FILLING_STATE := E_MET_CRYO_LN2_FILLING_STATE.NONE; // Used in case we restart in shields already cold
	
	nPTCStartingState:  UINT := 0;
	nPTCTempCtrlState:  UINT := 0;
	nStopCoolDownState:  UINT := 0;	
END_STRUCT
END_TYPE

// DUTs/Structures/Routines/Cool_Down/T_MET_CRYO_COOLDOWN_SYS_INPUT
// NOTE: Not used yet !!!
// Should replace input parameters of FB_CRYO_EVACUATION_SYSTEM.
// Should be set with NEW method FB_CRYO_CTRL::M_SetEvacSystemInputData().
TYPE T_MET_CRYO_COOLDOWN_SYS_INPUT :
STRUCT
	//
	// System configuration
	//
	// Time between closing Vac valve and Switching OFF the vac Pump [ms]
	//nTime_DeltaTValve:		UDINT;	
	// Time [ms] to run Turbo Pump to consider vacuum is good (useful when cryostat is cold)
	//nTime_TurboPump:		UDINT;	

	lrPress_Atm:			LREAL;	// Atmospheric pressure limit   [mbar]

	//lrTemp_Precooled:		LREAL;	// Precooled temperature limit [K]
	lrTemp_Warm:			LREAL;	// Warm      temperature limit [K]

	//
	// System configuration
	//
	lrTemp_Cryo:			T_CRYO_TEMPERATURE_STATUS;	// Cold Bench temperature	
	lrPressure_Cryo:		T_CRYO_PRESSURE_STATUS;		// Cryostat Pressure
	lrPressure_Evac:		T_CRYO_PRESSURE_STATUS;		// Evacuation Pressure
	bRepressValveOpen:		BOOL;	// Repressure Valve Open flag
	bRepressValveOK:		BOOL;	// Repressure Valve OK flag
END_STRUCT
END_TYPE

// DUTs/Structures/Routines/Cool_Down/T_MET_CRYO_COOLDOWN_SYSTEM_STATUS
TYPE T_MET_CRYO_COOLDOWN_SYSTEM_STATUS :
STRUCT
	bDone:			BOOL;			// Flag if controller is OK
	bBusy:			BOOL;			// Flag if controller is BUSY
	bEnabled:		BOOL := FALSE;	// Controller active while bEnable is TRUE
	bError:			BOOL;			// Flag if controller is OK
	bActive:		BOOL;			// Flag if controller is ACTIVE
	bEmergency:		BOOL := FALSE;	// Flag if there was Emergency valve closure
//	bRootPumpON:	BOOL;			// Flag if Root Pump is running
//	bTurboPumpON:	BOOL;			// Flag if Turbo Pump is running
//	bTurboPump10min:BOOL;			// Flag if Turbo Pump has been running for more than 10 min
	bValveOpen:		BOOL;			// Flag if Venting Valve is open

	// Generic controller OK flag.
	// Used for problems other than from the actuator.
	// This flag is used for problems coming from controllers
	// that extend the functionality of FB_CRYO_BIN_CTRL.
	bCtrlOK:	BOOL := TRUE;		

	nCycleCounter:	UDINT := 0;
	nLastCommand:	E_CRYO_BIN_ACT_CMD	:= E_CRYO_BIN_ACT_CMD.NONE;	// Command
	nState:			E_MET_CRYO_VENTING_SYS_STATE	:= E_MET_CRYO_VENTING_SYS_STATE.NONE;
	
	sState:			STRING(64);		// State as text
	sStatus:		STRING(64);		// Status as text
END_STRUCT
END_TYPE

// DUTs/Structures/Routines/Evacuation/T_MET_CRYO_EVACUATION_CTRL
TYPE T_MET_CRYO_EVACUATION_CTRL :
STRUCT
	{attribute 'TcHmiSymbol.Show'}
	bEnable:						BOOL := FALSE;
	bStop:							BOOL := FALSE;
	bReset:							BOOL := FALSE;
	
	por_VAGF1:	FB_CRYO_CMD_OVERRIDE;
	por_VAGF2:	FB_CRYO_CMD_OVERRIDE;
	por_VAGG1:	FB_CRYO_CMD_OVERRIDE;
	por_VAGG2:	FB_CRYO_CMD_OVERRIDE;
	por_VAGF:	FB_CRYO_CMD_OVERRIDE;
	por_VAGG:	FB_CRYO_CMD_OVERRIDE;
	
	bSim_Press_VAGF: 	BOOL;
	bSim_Press_VAGG: 	BOOL;
	
	bSim_Press_VAGF1: 	BOOL;
	bSim_Press_VAGF2: 	BOOL;
	bSim_Press_VAGG1: 	BOOL;
	bSim_Press_VAGG2: 	BOOL;

	
END_STRUCT
END_TYPE

// DUTs/Structures/Routines/Evacuation/T_MET_CRYO_EVACUATION_STAT
TYPE T_MET_CRYO_EVACUATION_STAT :
STRUCT
	bEnabled:		BOOL := FALSE;	// Controller active while bEnable is TRUE
	bConfigured:	BOOL := FALSE;	// Flag if controller has been configured.
	bError:			BOOL;			// Flag if controller is OK
	bActive:		BOOL;			// Flag if controller is ACTIVE
	bEmergency:		BOOL := FALSE;	// Flag if there was Emergency valve closure
	bInterlock:		BOOL := TRUE;	// Flag if there is an Interlock
	bDone:					BOOL;			// Flag if controller is OK
	bBusy:					BOOL;			// Flag if controller is BUSY
	bAlarm:					BOOL := FALSE;
	bWarning:				BOOL := FALSE;
	bPreConditionsMet:		BOOL := FALSE;
	{attribute 'TcHmiSymbol.Show'}	
	bAuto:					BOOL := TRUE;
	{attribute 'TcHmiSymbol.Show'}
	bManual:				BOOL := FALSE;
	
	//bRootPumpON:	BOOL;			// Flag if Root Pump is running
	//bTurboPumpON:	BOOL;			// Flag if Turbo Pump is running
//	bN2C1Open:		BOOL;			// Flag if venting N2C_1 valve is open
//	bN2C2Open:		BOOL;			// Flag if venting N2C_1 valve is open
	bVentingValvesOpen:		BOOL;	// Flag if all venting valves are open
//	bValveAfterTP:	BOOL := FALSE;	// Flag if Evacuation Valve should open after TP has started

	// Generic controller OK flag.
	// Used for problems other than from the actuator.
	// This flag is used for problems coming from controllers
	// that extend the functionality of FB_CRYO_BIN_CTRL.
	bCtrlOK:	BOOL := TRUE;		

	nCycleCounter:	UDINT := 0;
	nState:			E_MET_CRYO_VENTING_STATE	:= E_MET_CRYO_VENTING_STATE.NONE;
	
	sErrorText:		STRING(64);		// Error as text
	{attribute 'TcHmiSymbol.Show'}
	sState:			STRING(64);		// State as text
	sStatus:		STRING(64);		// Status as text
	
	// Error handeling	

	Error: 		T_METIS_CRYO_ERROR_STATUS;
	sErrorMessage:		STRING(256) := '';		// Error message	
	nErrorCode:			UDINT := 0;
	sRecoverySuggestion: STRING(256) := '';
	
END_STRUCT
END_TYPE

// DUTs/Structures/Routines/Re_Generation/T_MET_CRYO_RE_GENERATION_CTRL
TYPE T_MET_CRYO_RE_GENERATION_CTRL :
STRUCT

	bEnable:						BOOL := FALSE;
	bReset:							BOOL := FALSE;
	
END_STRUCT
END_TYPE

// DUTs/Structures/Routines/Re_Generation/T_MET_CRYO_RE_GENERATION_STAT
TYPE T_MET_CRYO_RE_GENERATION_STAT :
STRUCT
	
	bEnabled:				BOOL := FALSE;	// Controller active while bEnable is TRUE
	bConfigured:			BOOL := FALSE;	// Flag if controller has been configured.
	bError:					BOOL;			// Flag if controller is OK
	bActive:				BOOL;			// Flag if controller is ACTIVE
	bDone:					BOOL;			// Flag if controller is OK
	bBusy:					BOOL;			// Flag if controller is BUSY
	bAlarm:					BOOL := FALSE;
	bWarning:				BOOL := FALSE;
	
	bReadyToEnable:			BOOL := FALSE;
	bReadyToDisable:		BOOL := FALSE;
	bPreConditionsMet:		BOOL := FALSE;
	
	nState: E_MET_CRYO_RE_GENERATION_STATE := E_MET_CRYO_RE_GENERATION_STATE.NONE;
	sState:					STRING(80) := 'OFF';
	sErrorText:				STRING(64);		// Error as text
	
	bPermitEvacuationStop:	BOOL := TRUE;
	
	// Error handeling	

	Error: 		T_METIS_CRYO_ERROR_STATUS;
	sErrorMessage:		STRING(256) := '';		// Error message	
	nErrorCode:			UDINT := 0;
	sRecoverySuggestion: STRING(256) := '';
	
	
END_STRUCT
END_TYPE

// DUTs/Structures/Routines/Venting/T_MET_CRYO_VENTING_CFG
TYPE T_MET_CRYO_VENTING_CFG :
STRUCT

	nType_HPG1:		E_CRYO_SENSOR_TYPE_PRESS := E_CRYO_SENSOR_TYPE_PRESS.CMR_361;
	nType_HPG2:		E_CRYO_SENSOR_TYPE_PRESS := E_CRYO_SENSOR_TYPE_PRESS.CMR_361;	
	
	tDelay:		TIME := T#3S;	// Time delay before stopping Turbo Pump
	
	tWaitingTimeToStartVenting:	TIME := T#30S; // Waiting time after Enabling Venting
	
	(* *)
	lrMaxVentingPressure:	LREAL := 1060; // HPG = P ambient + 50 mbar 
	
	
	
END_STRUCT
END_TYPE

// DUTs/Structures/Routines/Venting/T_MET_CRYO_VENTING_CTRL
TYPE T_MET_CRYO_VENTING_CTRL :
STRUCT

	bEnable:						BOOL := FALSE;
	bStop:							BOOL := FALSE;
	bReset:							BOOL := FALSE;
	bEnable_N2V_1:	BOOL := FALSE;
	bEnable_N2V_2:	BOOL := FALSE;

	// Override flags	
	// Valve command override handling
	cor_N2V_1:	FB_CRYO_CMD_OVERRIDE;
	cor_N2V_2:	FB_CRYO_CMD_OVERRIDE;

// HPG pressure override	
	por_HPG:	FB_CRYO_CMD_OVERRIDE;
	bSim_Press_HPG: 	BOOL;
	
	por_HPG1:	FB_CRYO_CMD_OVERRIDE;
	bSim_Press_HPG1: 	BOOL;
	
	por_HPG2:	FB_CRYO_CMD_OVERRIDE;
	bSim_Press_HPG2: 	BOOL;
	
END_STRUCT
END_TYPE

// DUTs/Structures/Routines/Venting/T_MET_CRYO_VENTING_STAT
TYPE T_MET_CRYO_VENTING_STAT :
STRUCT
	bEnabled:		BOOL := FALSE;	// Controller active while bEnable is TRUE
	bConfigured:	BOOL := FALSE;	// Flag if controller has been configured.
	bError:			BOOL;			// Flag if controller is OK
	bActive:		BOOL;			// Flag if controller is ACTIVE
	bEmergency:		BOOL := FALSE;	// Flag if there was Emergency valve closure
	bDone:					BOOL;			// Flag if controller is OK
	bBusy:					BOOL;			// Flag if controller is BUSY
	bAlarm:					BOOL := FALSE;
	bWarning:				BOOL := FALSE;
	bPreConditionsMet:		BOOL := FALSE;
		
	bN2C1Open:		BOOL;			// Flag if venting N2C_1 valve is open
	bN2C2Open:		BOOL;			// Flag if venting N2C_1 valve is open
	bVentingValvesOpen:		BOOL;	// Flag if all venting valves are open
//	bValveAfterTP:	BOOL := FALSE;	// Flag if Evacuation Valve should open after TP has started

	// Generic controller OK flag.
	// Used for problems other than from the actuator.
	// This flag is used for problems coming from controllers
	// that extend the functionality of FB_CRYO_BIN_CTRL.
	bCtrlOK:	BOOL := TRUE;		

	nCycleCounter:	UDINT := 0;
	nState:			E_MET_CRYO_VENTING_STATE	:= E_MET_CRYO_VENTING_STATE.NONE;
	
	sErrorText:		STRING(64);		// Error as text
	sState:			STRING(64);		// State as text
	sStatus:		STRING(64);		// Status as text
	
	bVentingPressureAchieved:	BOOL := FALSE;
	
	// Error handeling	

	Error: 		T_METIS_CRYO_ERROR_STATUS;
	sErrorMessage:		STRING(256) := '';		// Error message	
	nErrorCode:			UDINT := 0;
	sRecoverySuggestion: STRING(256) := '';
	
	
END_STRUCT
END_TYPE

// DUTs/Structures/Routines/Venting/T_MET_CRYO_VENTING_SYS_INPUT
// NOTE: Not used yet !!!
// Should replace input parameters of FB_CRYO_EVACUATION_SYSTEM.
// Should be set with NEW method FB_CRYO_CTRL::M_SetEvacSystemInputData().
TYPE T_MET_CRYO_VENTING_SYS_INPUT :
STRUCT
	//
	// System configuration
	//
	// Time between closing Vac valve and Switching OFF the vac Pump [ms]
	//nTime_DeltaTValve:		UDINT;	
	// Time [ms] to run Turbo Pump to consider vacuum is good (useful when cryostat is cold)
	//nTime_TurboPump:		UDINT;	

	lrPress_Atm:			LREAL;	// Atmospheric pressure limit   [mbar]

	//lrTemp_Precooled:		LREAL;	// Precooled temperature limit [K]
	lrTemp_Warm:			LREAL;	// Warm      temperature limit [K]

	//
	// System configuration
	//
	lrTemp_Cryo:			T_CRYO_TEMPERATURE_STATUS;	// Cold Bench temperature	
	lrPressure_Cryo:		T_CRYO_PRESSURE_STATUS;		// Cryostat Pressure
	lrPressure_Evac:		T_CRYO_PRESSURE_STATUS;		// Evacuation Pressure
	bRepressValveOpen:		BOOL;	// Repressure Valve Open flag
	bRepressValveOK:		BOOL;	// Repressure Valve OK flag
END_STRUCT
END_TYPE

// DUTs/Structures/Routines/Venting/T_MET_CRYO_VENTING_SYSTEM_STATUS
TYPE T_MET_CRYO_VENTING_SYSTEM_STATUS :
STRUCT
	bDone:			BOOL;			// Flag if controller is OK
	bBusy:			BOOL;			// Flag if controller is BUSY
	bEnabled:		BOOL := FALSE;	// Controller active while bEnable is TRUE
	bError:			BOOL;			// Flag if controller is OK
	bActive:		BOOL;			// Flag if controller is ACTIVE
	bEmergency:		BOOL := FALSE;	// Flag if there was Emergency valve closure
//	bRootPumpON:	BOOL;			// Flag if Root Pump is running
//	bTurboPumpON:	BOOL;			// Flag if Turbo Pump is running
//	bTurboPump10min:BOOL;			// Flag if Turbo Pump has been running for more than 10 min
	bValveOpen:		BOOL;			// Flag if Venting Valve is open

	// Generic controller OK flag.
	// Used for problems other than from the actuator.
	// This flag is used for problems coming from controllers
	// that extend the functionality of FB_CRYO_BIN_CTRL.
	bCtrlOK:	BOOL := TRUE;		

	nCycleCounter:	UDINT := 0;
	nLastCommand:	E_CRYO_BIN_ACT_CMD	:= E_CRYO_BIN_ACT_CMD.NONE;	// Command
	nState:			E_MET_CRYO_VENTING_SYS_STATE	:= E_MET_CRYO_VENTING_SYS_STATE.NONE;
	
	sState:			STRING(64);		// State as text
	sStatus:		STRING(64);		// Status as text
END_STRUCT
END_TYPE

// DUTs/Structures/Routines/WarmUp/T_MET_CRYO_WARMUP_CTRL
TYPE T_MET_CRYO_WARMUP_CTRL :
STRUCT

	bEnable:						BOOL := FALSE;
	bStop:							BOOL := FALSE;
	bReset:							BOOL := FALSE;
	
END_STRUCT
END_TYPE

// DUTs/Structures/Routines/WarmUp/T_MET_CRYO_WARMUP_STAT
TYPE T_MET_CRYO_WARMUP_STAT :
STRUCT
	

	bEnabled:				BOOL := FALSE;	// Controller active while bEnable is TRUE
	bConfigured:			BOOL := FALSE;	// Flag if controller has been configured.
	bError:					BOOL;			// Flag if controller is OK
	bActive:				BOOL:= FALSE;			// Flag if controller is ACTIVE
	bDone:					BOOL;			// Flag if controller is OK
	bBusy:					BOOL;			// Flag if controller is BUSY
	bAlarm:					BOOL := FALSE;
	bWarning:				BOOL := FALSE;
	
	bEmergency:				BOOL := FALSE;	// Flag if there was Emergency valve closure
	bPreConditionsMet:		BOOL := FALSE;

	nState:			E_MET_CRYO_WARMUP_STATE	:= E_MET_CRYO_WARMUP_STATE.NONE;
	
	
	sState:			STRING(64);		// State as text
	sStatus:		STRING(64);		// Status as text
	sErrorText:		STRING(64);		// Error as text
	
	bPermitEvacuationStop:			BOOL := TRUE;
	bPermitVenting:					BOOL := TRUE;
	
	// Error handeling	

	Error: 		T_METIS_CRYO_ERROR_STATUS;
	sErrorMessage:		STRING(256) := '';		// Error message	
	nErrorCode:			UDINT := 0;
	sRecoverySuggestion: STRING(256) := '';
	
	
	
END_STRUCT
END_TYPE

// DUTs/Structures/Sensors/LN2_Level_Sensor/T_METIS_CRYO_LN2_LEVEL_CFG
TYPE T_METIS_CRYO_LN2_LEVEL_CFG :
STRUCT
//	// Threshold temperature read by the heated pt100s when submerged under LN2
//		lrLN2_Level_SenseTempK_HA:		LREAL := 90.0;
//		lrLN2_Level_SenseTempK_H:		LREAL := 85.0;
//		lrLN2_Level_SenseTempK_L:		LREAL := 85.0;
//		lrLN2_Level_SenseTempK_LA:		LREAL := 85.0;

//	// Threshold temperature read by the heated pt100s when LN2 is absent OR Evaporated 
		
//		lrLN2_Level_AbsenceTempK_HA:	LREAL := 90.0;
//		lrLN2_Level_AbsenceTempK_H:		LREAL := 85.0;
//		lrLN2_Level_AbsenceTempK_L:		LREAL := 85.0;
//		lrLN2_Level_AbsenceTempK_LA:	LREAL := 85.0;
		
		
		 
END_STRUCT
END_TYPE

// DUTs/Structures/Sensors/LN2_Level_Sensor/T_METIS_CRYO_LN2_LEVEL_STATUS
{attribute 'TcHmiSymbol.Show'}
TYPE T_METIS_CRYO_LN2_LEVEL_STATUS :
STRUCT
	{attribute 'TcHmiSymbol.Show'}
	{attribute 'TcHmiSymbol.ReadOnly'}
	bSimulated:		BOOL;				// Flag indicating if the value is simulated.
	{attribute 'TcHmiSymbol.Show'}
	{attribute 'TcHmiSymbol.ReadOnly'}
	lrSimTempK:		LREAL;				// Simulated temperature value in [K].
	{attribute 'TcHmiSymbol.Show'}
	{attribute 'TcHmiSymbol.ReadOnly'}
	bValid:			BOOL	:= FALSE;	
	{attribute 'TcHmiSymbol.Show'}
	{attribute 'TcHmiSymbol.ReadOnly'}
	bHighAlarm:		BOOL	:= FALSE;
	{attribute 'TcHmiSymbol.Show'}
	{attribute 'TcHmiSymbol.ReadOnly'}
	bHigh:			BOOL	:= FALSE;
	{attribute 'TcHmiSymbol.Show'}
	{attribute 'TcHmiSymbol.ReadOnly'}
	bLow:			BOOL	:= FALSE;
	{attribute 'TcHmiSymbol.Show'}
	{attribute 'TcHmiSymbol.ReadOnly'}
	bLowAlarm:		BOOL	:= FALSE;
	{attribute 'TcHmiSymbol.Show'}
	{attribute 'TcHmiSymbol.ReadOnly'}
	bLN2_Supply_Empty:	BOOL	:= FALSE;	// LN2 not present if all LN2 levels are FALSE
	{attribute 'TcHmiSymbol.Show'}
	{attribute 'TcHmiSymbol.ReadOnly'}
	bActive:		BOOL	:= TRUE;	// Level Sensor is active when heater are enabled 
	

	
	
//	bInRange:		BOOL	:= FALSE;
	{attribute 'TcHmiSymbol.Show'}
	{attribute 'TcHmiSymbol.ReadOnly'}
	bWarningSens_HA:	BOOL	:= TRUE;
	{attribute 'TcHmiSymbol.Show'}
	{attribute 'TcHmiSymbol.ReadOnly'}
	bWarningSens_H:		BOOL	:= TRUE;
	{attribute 'TcHmiSymbol.Show'}
	{attribute 'TcHmiSymbol.ReadOnly'}
	bWarningSens_L:		BOOL	:= TRUE;
	{attribute 'TcHmiSymbol.Show'}
	{attribute 'TcHmiSymbol.ReadOnly'}
	bWarningSens_LA:	BOOL	:= TRUE;
	{attribute 'TcHmiSymbol.Show'}
	{attribute 'TcHmiSymbol.ReadOnly'}
	bError:				BOOL	:= TRUE;
	{attribute 'TcHmiSymbol.Show'}
	{attribute 'TcHmiSymbol.ReadOnly'}
	sStatus:			STRING	:= '';
	{attribute 'TcHmiSymbol.Show'}
	{attribute 'TcHmiSymbol.ReadOnly'}
	sName:			STRING	:= '';


//	lrRamp:			LREAL;				// Temperature ramp [deg/min]
//	lrTempC:		LREAL;				// Temp [deg C]
//	lrTempK:		LREAL;				// Temp [deg K]
END_STRUCT
END_TYPE

// DUTs/Structures/System/T_METIS_CRYO_CFG
TYPE T_METIS_CRYO_CFG :
STRUCT
	

	lrTemp_Cold:			LREAL := 75.0;	// Cool      temperature limit [K] = 10 C
	lrTemp_OP:				LREAL := 60.0;	// Operational temperature limit [K]
	lrTemp_Warm:			LREAL := 285.0;	// Warm      temperature limit [K] = 20 C
	lrTempColdRadShield:	LREAL := 100.0; // Radiation shield temps at COLD state
	
	lrTemp_Preamp:			LREAL := 120.0;	// Heater preemp target temperature [K]
	lrTemp_LowLimit:		LREAL :=  73.0;	// Lowest    temperature limit [K]
	
	tInitTimeOut:			TIME  := T#60S;
	
	
	lrVaccum_To_Start_CoolDown: LREAL := 0.0001; // p < 1e-4 mbar 
	lrVaccum_Press_Operations:		 			LREAL := 0.00001; // p < 1e-6 mbar 
	lrLow_Vacuum_Press_Warning_For_Operations: 	LREAL := 0.00001; // TBC ?? 
	lrLow_Vacuum_Press_Alarm_For_Operations: 	LREAL := 0.00001; // TBC ??
	


	/////////////
	// Cool-Down//
	////////////
	
	lrCoolDown_PreCond_Press:			LREAL := 0.0001; // p<1e-4 mbar pressure
	lrCoolDown_LN2_TempK:				LREAL := 100;    // 100 K temp threshold
	lrRadShld_TempK_TO_Start_PTCs: 		LREAL := 120; // 
	
	/////////////
	// Warm_UP//
	////////////
	lrWarmUp_Detectors_Ramp_1:				LREAL := 1.0; // Start detectors warm up with a ramp of 1 K/min
	lrWarmUp_Detectors_Ramp_Switch_Temp:	LREAL := 80.0; // ramp switch at 80 K from 1K/min to 6K/h
	lrWarmUp_Detectors_Ramp_2:				LREAL := 0.1; // ramp up detectors, new ramp 6 K/h (0.1 K/min)
	lrWarmUp_EvacPermission_Temp:			LREAL := 280; // When all temperatures > 280 K,  allow to stop evacuation
	lrWarmUp_VentingPermission_Temp:		LREAL := 280; // When all temperatures > 280 K, allow tO start venting routine 
	lrWarmUp_Alarm_Temp:					LREAL := 310; 
	lrWarmUp_Alarm_PreCooling_Pressure:		LREAL := 700; // Pressure precooling system >700 mbar
	// TODO: Detector ramp too fast
	
	///////////////////	
	// Re_Generation//
	//////////////////
	lrRegeneration_Safe_Temp:			LREAL := 280.0;   // All temperatures above 280 K before Regeneration can begin 
	lrRegeneration_Safe_Press:			LREAL := 0.01;
	lrTemp_Regeneration_SetPoint: 		LREAL := 333.0; // Regeneration heater setpoint[K]
	lrTemp_Regeneration_Alarm_Temp:		LREAL := 340.0;	// Alarm when t_sorption_pump > 340 [K]
	lrTemp_Regeneration_Alarm_Press:	LREAL := 0.01;	// Alarm when	Pressure inside cryostat > 1e-2 mbar
	lrTemp_Regeneration_Stop:			LREAL := 310.0; // After sorption cool_down, once it reaches 310, safe to stop Regeneration and Evac
	tSorption_Pump_Cool_Down_TimeOut: 	TIME  := T#3H;   // Time after sorption pump heaters are OFF

	///////////////////	
	// Anti-Fogging //
	//////////////////
	
	lrAntiFog_Purging_DewPoint:			LREAL := 10.0; // If dew-point is <10 K below ambient window purging is started
	lrAntiFog_Heating_DewPoint:			LREAL := 10.0; // If dew-point is <5 K below ambient window increased window heating is started
	lrAntiFog_DewPoint_Alarm:			LREAL := 5.0;  // dew point is <5 K below window temperature
	
	

	lrPress_Atm:			LREAL := 1000;		// Atmospheric pressure limit   [mbar]
	lrPress_InVac:			LREAL := 10.0E-4;	// In vacuum limit   [mbar]
	lrPress_GoodVac:		LREAL := 10.0E-6;	// Good Vacuum limit [mbar]
	
	

END_STRUCT
END_TYPE

// DUTs/Structures/System/T_METIS_CRYO_CTRL
TYPE T_METIS_CRYO_CTRL :
STRUCT
	bExecute:	BOOL := FALSE;
	nCommand:	E_METIS_CRYO_CTRL_CMD := E_METIS_CRYO_CTRL_CMD.NONE;
	
	bReset:		BOOL := FALSE;		// RESET Command
	
	bInitialize: BOOL := FALSE; 	// Initailaze the higher level control
	bEnable:	 BOOL := FALSE;

//	// Command to repressurize the system. 
//	// Exists only in full simulation in order to bring the 
//	// system to atmospheric pressure.
//	// In reality, repressurization is done by opening a manual valve.
//	bSim_Repress:	BOOL := FALSE;	

	//
	// Enable flags used to activate system functions. 	
	//
	{attribute 'TcHmiSymbol.Show'}
	bEnable_Evac:				BOOL := FALSE;
	bEnable_Cool_Down:			BOOL := FALSE;
	bEnable_Stop_Cool_Down:		BOOL := FALSE;
	bEnable_Warm_Up:			BOOL := FALSE;
	bEnable_Regeneration:		BOOL := FALSE;
	bEnable_Anti_Fogging:		BOOL := FALSE;
	bEnable_Power_Outage:		BOOL := FALSE;
	bEnable_Stop_Power_Outage:	BOOL := FALSE;
	
	bEnable_Venting:			BOOL := FALSE;
	

	//	
	// Safe flags saying what is safe and what not.
	//
	bSafe_Evac:					BOOL := FALSE;
	bSafe_Cool_Down:			BOOL := FALSE;
	bSafe_Stop_Cool_Down:		BOOL := FALSE;
	bSafe_Warm_Up:				BOOL := FALSE;
	bSafe_Regeneration:			BOOL := FALSE;
	bSafe_Anti_Fogging:			BOOL := FALSE;
//	bSafe_Power_Outage:			BOOL := FALSE;
//	bSafe_Stop_Power_Outage:	BOOL := FALSE;
	
	bSafe_Venting:	BOOL := FALSE;
	
	
	// Coolant Valves
	bEnable_TPC_A:	BOOL := FALSE;
	bEnable_TPC_B:	BOOL := FALSE;
	
	cor_TPC_A:	FB_CRYO_CMD_OVERRIDE;
	cor_TPC_B:	FB_CRYO_CMD_OVERRIDE;
	
// Coolers

	// Sleeves Pressures overrides	
	por_VAG_PTA:	FB_CRYO_CMD_OVERRIDE;
	bSim_Press_VAG_PTA: 	BOOL;
	
	por_VAG_PTB:	FB_CRYO_CMD_OVERRIDE;
	bSim_Press_VAG_PTB: 	BOOL;
	
	por_VAG_PTC:	FB_CRYO_CMD_OVERRIDE;
	bSim_Press_VAG_PTC: 	BOOL;

	
END_STRUCT
END_TYPE

// DUTs/Structures/System/T_METIS_CRYO_DEBUG
TYPE T_METIS_CRYO_DEBUG :
STRUCT
	nCycleCounter:	UDINT := 0;
END_STRUCT
END_TYPE

// DUTs/Structures/System/T_METIS_CRYO_EVENTS
TYPE T_METIS_CRYO_EVENTS :
STRUCT
//	info:		FB_TcMessage;
//	warning:	FB_TcMessage;
//	error:		FB_TcAlarm;
//	critical:	FB_TcAlarm;
	
END_STRUCT
END_TYPE

// DUTs/Structures/System/T_METIS_CRYO_INTERLOCKS
TYPE T_METIS_CRYO_INTERLOCKS :
STRUCT
	bInterlock_Evacuation:		BOOL := FALSE;
	bInterlock_Venting:			BOOL := FALSE;
	bInterlock_CoolDown:		BOOL := FALSE;
	bInterlock_WarmUp:			BOOL := FALSE;
	bInterlock_Regeneration:	BOOL := FALSE;
	bInterlock_AntiFogging:		BOOL := FALSE;
	bInterlock_PowerOutage:		BOOL := FALSE;
	bInterlock_StopPowerOutage:	BOOL := FALSE;
	sInterlockState:			STRING := 'Initializing';
END_STRUCT
END_TYPE

// DUTs/Structures/System/T_METIS_CRYO_STAT
TYPE T_METIS_CRYO_STAT :
STRUCT
	//
	// Common attributes
	//
	bConfigured:	BOOL := FALSE;
	bInitialized:   BOOL := FALSE;
	//
	bSystemStarted:	BOOL := FALSE;	// Indicates if M_GetState has been called.
	bDone:			BOOL;			// Flag if controller is OK
	bBusy:			BOOL;			// Flag if controller is BUSY
	bError:			BOOL;			// Flag if controller is OK
	bActive:		BOOL;			// Flag if controller is ACTIVE
	
	bAlarm:			BOOL;			// 
	bWarning:		BOOL;
	
	bSimulation:	BOOL := FALSE; // simlation active when version V2_SIM is active
	
//	nLastCommand:	E_PDS_CRYO_CTRL_CMD 	:= E_PDS_CRYO_CTRL_CMD.NONE;
//	nState:			E_PDS_CRYO_CTRL_STATE	:= E_PDS_CRYO_CTRL_STATE.NONE;
	sState:			STRING(64);		// State as text
	
	// Generic controller OK flag.
	// Used for problems other than from the actuator.
	// This flag is used for problems coming from controllers
	// that extend the functionality of FB_CRYO_BIN_CTRL.
	bCtrlOK:		BOOL := TRUE;	

	bSafeToDisableSystem:	BOOL := FALSE;	

	// Routine Status

	bEvacuationActive:		BOOL := FALSE;
	bVentingActive:			BOOL := FALSE;
	bCoolDownActive:		BOOL := FALSE;
	bWarmUpActive:			BOOL := FALSE;
	bRegenerationActive:	BOOL := FALSE;
	bAntiFoggingActive:		BOOL := FALSE;
	bPowerOutageActive:		BOOL := FALSE;
	bStopPowerOutageActive:	BOOL := FALSE;
	
	// 
	bVentingFinishedSuccessfully: BOOL := FALSE;
	// 
	lrVAGF:			LREAL;
	lrVAGG:			LREAL;
	lrHPG:			LREAL;
	lrCryoPressure: 		LREAL; // TBC ??
	bCryoPressureValid:		BOOL := FALSE;
	
	bPressurized:	BOOL := FALSE;	
	bPartialVacuum:	BOOL := FALSE;
	bInVacuum:		BOOL := FALSE;	
	bInGoodVacuum:	BOOL := FALSE;  // To 1e-6 mbar
 		
	bWarm:			BOOL := FALSE;
	bPartiallyCold:	BOOL := FALSE;
	bCold:			BOOL := FALSE;	// Master temperature < cfg.lrTemp_Cold		??
	bOP:			BOOL := FALSE;	// Master temperature < cfg.lrTemp_OP		??
	

	bCoolantFlowOK:	BOOL := FALSE;		


	
	// Statuses of critical devices
	
	bVentingValvesAreClosed:		BOOL := FALSE;
	bPumpsAreRunning:				BOOL := FALSE;
	bRoughingPumpsAreRunning:		BOOL := FALSE;
	bTurboPumpsRunning:				BOOL := FALSE;
	bWarmUpHeatersActive:			BOOL := TRUE;
	
	bManualValvesAreClosed:			BOOL := FALSE;
	
	bDetectorTempSafe:				BOOL := FALSE;
	
	////
	lrDewPointTempC:					LREAL;
	lrAmbiantTempC:						LREAL;
	lrWindowMountTempC:					LREAL;
	
	lrDewPointTempK:					LREAL;
	lrAmbiantTempK:						LREAL;
	lrWindowMountTempK:					LREAL;	
	
	// Detector Temp. and Heater statuses


	//
	// Temperatures [K]
	//
	
	lrRadShieldStiffRingTempK:			LREAL; // Temp vote of which temp sensors? TBC
	lrRadShieldIntermediateTempK:			LREAL; // Temp vote of which temp sensors? TBC
	lrRadShieldBottomTempK:			LREAL; // Temp vote of which temp sensors? TBC
	lrRadiationShieldsTempK:			LREAL; // Average temperature of all radiation shields
	
	
	// TODO: Link to ptoper sensor
	bHighestTempValid:	BOOL := TRUE;	// Highest temperature Valid flag
	bLowestTempValid:	BOOL := TRUE;	// Lowest temperature Valid flag

	lrHighestTempK:	LREAL;	// Highest temperature [K] in Cryostat
	lrLowestTempK:	LREAL;	// Lowest temperature [K] in Cryostat
	
	sHighestTempName:	STRING;
	sLowestTempName:	STRING;
	
	lrAverageOfAllTemps: LREAL;

	// TODO: link to an appropriate T-vote
	lrCryoTempK:		LREAL := 281.0; // Cryostat temperature 
	
	// Stop PTCs during Warm_Up
	bStop_PTCs:			BOOL := TRUE;

	// Permission from different procedure to stop the Evacuation

	bPermitEvacuationStop: BOOL := FALSE;
	 
	nCycleCounter:	UDINT := 0; 
	nLastCommand:	E_METIS_CRYO_CTRL_CMD 	:= E_METIS_CRYO_CTRL_CMD.NONE;
	nState:			E_METIS_CRYO_CTRL_STATE	:= E_METIS_CRYO_CTRL_STATE.NONE;
	
	// N2 Gas supply Connected for Cryostat venting
	bGN2SupplyConnected:	BOOL := TRUE;

		// Error handeling	

	Error: 		T_METIS_CRYO_ERROR_STATUS;
	sErrorMessage:		STRING(256) := '';		// Error message	
	nErrorCode:			UDINT := 0;
	sRecoverySuggestion: STRING(256) := '';
	
	// Ambient Pressure [mbar]
	lrAmbientPressure:		LREAL;
	
END_STRUCT
END_TYPE

// DUTs/Structures/System/T_METIS_CRYO_TRIGGERS
TYPE T_METIS_CRYO_TRIGGERS :
STRUCT
	//
	// Evacuation pumps
	//
	PVV1_Open:		R_TRIG;	// evac.PVV1.in_bEnable
	PVV1_Close:		F_TRIG;	// evac.PVV1.in_bEnable
	PVV1_Opened:	R_TRIG;	// evac.PVV1.stat.bActON
	PVV1_Closed:	R_TRIG;	// evac.PVV1.stat.bActOFF

	PVP_Start:		R_TRIG;	// evac.pump_pvp.in_bEnable
	PVP_Stop:		F_TRIG;	// evac.pump_pvp.in_bEnable
	PVP_Ready:		R_TRIG;	// evac.pump_pvp.stat.bReady
	PVP_Stopped:	F_TRIG;	// evac.pump_pvp.stat.bMoving

	//
	// Evacuation valve
	//
	TMP_Start:		R_TRIG;	// evac.pump_tmp.in_bEnable
	TMP_Stop:		F_TRIG;	// evac.pump_tmp.in_bEnable
	TMP_Ready:		R_TRIG;	// evac.pump_tmp.stat.bReady
	TMP_Stopped:	F_TRIG;	// evac.pump_tmp.stat.bMoving
	
	//
	// Heaters
	//
	Heater_DetIF_Enable:		R_TRIG;	// Heater_DetIF.in_bEnable
	Heater_DetIF_Disable:		F_TRIG;	// Heater_DetIF.in_bEnable
	Heater_DetIF_ON:			R_TRIG;	// Heater_DetIF.stat.bActON
	Heater_DetIF_OFF:			R_TRIG;	// Heater_DetIF.stat.bActOFF

	Heater_Preamp_Enable:		R_TRIG;	// Heater_Preamp.in_bEnable
	Heater_Preamp_Disable:		F_TRIG;	// Heater_Preamp.in_bEnable
	Heater_Preamp_ON:			R_TRIG;	// Heater_Preamp.stat.bActON
	Heater_Preamp_OFF:			R_TRIG;	// Heater_Preamp.stat.bActOFF

	Heater_ColdPlate_Enable:	R_TRIG;	// Heater_ColdPlate.in_bEnable
	Heater_ColdPlate_Disable:	F_TRIG;	// Heater_ColdPlate.in_bEnable
	Heater_ColdPlate_ON:		R_TRIG;	// Heater_ColdPlate.stat.bActON
	Heater_ColdPlate_OFF:		R_TRIG;	// Heater_ColdPlate.stat.bActOFF

	//
	// Cooler
	//
	Cooler_Enable:		R_TRIG;	// cooler.in_bEnable
	Cooler_Disable:		F_TRIG;	// cooler.in_bEnable
	Cooler_ON:			R_TRIG;	// cooler.stat.nDevState
	Cooler_OFF:			R_TRIG;	// cooler.stat.nDevState


	//
	// Pressure and Temperature status flags
	//
	
	// Vacuum
	Vacuum_ON:		R_TRIG;	// stat.bInVacuum
	Vacuum_OFF:		F_TRIG;	// stat.bInVacuum
	Vacuum_OK:		R_TRIG;	// stat.bGoodVacuum
	Vacuum_NOT_OK:	F_TRIG;	// stat.bGoodVacuum

	// Temperature
	Cold_ON:		R_TRIG;	// stat.bCold
	Cold_OFF:		F_TRIG;	// stat.bCold
	OP_ON:			R_TRIG;	// stat.bOP
	OP_OFF:			F_TRIG;	// stat.bOP
	
END_STRUCT
END_TYPE

// DUTs/Structures/Temp_Sensor/T_METIS_DT670_TEMP_SENSOR_STATUS
TYPE T_METIS_DT670_TEMP_SENSOR_STATUS :
STRUCT
	//
	// Status coming from the analog input terminal.
	// This is nothing to do with the sensor, i.e. the reading can be
	// inside the input terminal measuring range but still it might
	// not be inside the sensor measuring range!
	//
	bInputUnder:		BOOL;
	bInputOver:			BOOL;
	bInputError:		BOOL;
	bInputToggle:		BOOL;
	bInputValid:		BOOL;
	bInputActive:		BOOL	:= FALSE;
	
	bLowWarning:		BOOL;
	bLowLowAlarm:		BOOL;
	bHighWarning:		BOOL;
	bHighHighAlarm:		BOOL;
	
	sErrorText:			STRING;
	
	lrRawValue:			LREAL;

	// Calculated status of the sensor
	bError:				BOOL;
	bWarning:			BOOL;
	bValid:				BOOL;
	
	sName:				STRING; // Sensor name
	sType:				STRING := 'DT670';
	
	nLSType:			E_METIS_LAKE_SHORE_TYPE;
	
	lrRamp:		LREAL;	// Temperature ramp [deg/min]
	lrTempC:	LREAL;	// Temperature in deg C
	lrTempK:	LREAL;	// Temperature in deg K
END_STRUCT
END_TYPE

// DUTs/Structures/Temp_Voter/T_HMI_METIS_TEMP_VOTER_CTRL
TYPE T_HMI_METIS_TEMP_VOTER_CTRL :
STRUCT
	mode      : E_HMI_CRYO_MODE := E_HMI_CRYO_MODE.NONE;
	eng       : E_HMI_CRYO_ENG := E_HMI_CRYO_ENG.NONE;
	sim_mode  : E_HMI_CRYO_SIMULATION_MODE_CTRL;
END_STRUCT
END_TYPE

// DUTs/Structures/Temp_Voter/T_HMI_METIS_TEMP_VOTER_STAT
TYPE T_HMI_METIS_TEMP_VOTER_STAT :
STRUCT
	temperature_stat : T_METIS_CRYO_TEMP_VOTE_STATUS;
	cmd_over_stat : T_HMI_CRYO_CMD_OVERRIDE_STAT;
END_STRUCT
END_TYPE

// DUTs/Structures/Temp_Voter/T_METIS_CRYO_TEMP_VOTE_STATUS
TYPE T_METIS_CRYO_TEMP_VOTE_STATUS :
STRUCT
	//
	// Status coming from the analog input terminal.
	// This is nothing to do with the sensor, i.e. the reading can be
	// inside the input terminal measuring range but still it might
	// not be inside the sensor measuring range!
	//
	bInputUnder:		BOOL;
	bInputOver:			BOOL;
	bInputError:		BOOL;
	bInputToggle:		BOOL;
	bInputValid:		BOOL;
	bInputActive:		BOOL	:= FALSE;
	nRawValue:			INT;

	// Calculated status of the sensor
	bError:				BOOL;
	
	{attribute 'TcHmiSymbol.Show'}
	{attribute 'TcHmiSymbol.ReadOnly'}
	lrRamp:		LREAL;	// Temperature ramp [deg/min]
	
